C09103=1053.163,-16.101,428.307,170.734,30.867,155.806
C09104=1053.169,-15.852,428.293,170.735,30.869,155.806
C09105=1053.175,-15.602,428.279,170.737,30.871,155.806
C09106=1053.182,-15.353,428.265,170.739,30.873,155.807
C09107=1053.188,-15.103,428.251,170.741,30.875,155.807
C09108=1053.194,-14.853,428.238,170.742,30.877,155.807
C09109=1053.200,-14.604,428.223,170.744,30.878,155.807
C09110=1053.206,-14.354,428.209,170.746,30.880,155.808
C09111=1053.213,-14.104,428.195,170.747,30.882,155.808
C09112=1053.218,-13.855,428.181,170.749,30.884,155.808
C09113=1053.224,-13.606,428.167,170.751,30.886,155.808
C09114=1053.231,-13.356,428.153,170.753,30.888,155.809
C09115=1053.236,-13.107,428.139,170.755,30.890,155.809
C09116=1053.243,-12.857,428.124,170.756,30.892,155.809
C09117=1053.249,-12.608,428.110,170.758,30.894,155.809
C09118=1053.255,-12.358,428.095,170.759,30.896,155.810
C09119=1053.261,-12.109,428.082,170.761,30.898,155.810
C09120=1053.268,-11.859,428.067,170.763,30.900,155.810
C09121=1053.274,-11.610,428.053,170.765,30.902,155.810
C09122=1053.280,-11.360,428.038,170.767,30.903,155.810
C09123=1053.286,-11.111,428.025,170.768,30.905,155.811
C09124=1053.297,-10.694,428.001,170.771,30.909,155.811
C09125=1053.307,-10.278,427.977,170.774,30.912,155.812
C09126=1053.317,-9.862,427.954,170.777,30.915,155.812
C09127=1053.327,-9.446,427.930,170.780,30.918,155.812
C09128=1053.334,-9.196,427.915,170.781,30.920,155.813
C09129=1053.339,-8.946,427.901,170.782,30.922,155.813
C09130=1053.346,-8.697,427.887,170.784,30.925,155.813
C09131=1053.352,-8.447,427.873,170.786,30.926,155.813
C09132=1053.358,-8.198,427.858,170.788,30.928,155.814
C09133=1053.365,-7.949,427.844,170.790,30.930,155.814
C09134=1053.371,-7.699,427.830,170.792,30.932,155.814
C09135=1053.377,-7.449,427.815,170.793,30.934,155.814
C09136=1053.384,-7.201,427.801,170.794,30.936,155.815
C09137=1053.390,-6.950,427.786,170.796,30.938,155.815
C09138=1053.396,-6.701,427.772,170.798,30.940,155.815
C09139=1053.402,-6.452,427.757,170.800,30.942,155.816
C09140=1053.409,-6.202,427.743,170.802,30.944,155.816
C09141=1053.415,-5.953,427.729,170.804,30.946,155.816
C09142=1053.421,-5.703,427.714,170.804,30.947,155.816
C09143=1053.426,-5.453,427.700,170.806,30.950,155.817
C09144=1053.434,-5.204,427.686,170.808,30.952,155.817
C09145=1053.440,-4.954,427.671,170.810,30.954,155.817
C09146=1053.445,-4.705,427.657,170.812,30.955,155.817
C09147=1053.453,-4.456,427.642,170.814,30.957,155.818
C09148=1053.459,-4.206,427.627,170.815,30.960,155.818
C09149=1053.464,-3.956,427.614,170.816,30.962,155.818
C09150=1053.471,-3.707,427.599,170.818,30.963,155.818
C09151=1053.478,-3.457,427.584,170.820,30.965,155.819
C09152=1053.486,-3.092,427.563,170.823,30.968,155.819
C09153=1053.496,-2.727,427.541,170.825,30.971,155.819
C09154=1053.504,-2.362,427.520,170.827,30.974,155.820
C09155=1053.513,-1.997,427.498,170.830,30.977,155.820
C09156=1053.519,-1.747,427.484,170.831,30.979,155.821
C09157=1053.525,-1.497,427.469,170.833,30.981,155.821
C09158=1053.531,-1.248,427.454,170.835,30.983,155.821
C09159=1053.537,-0.998,427.439,170.837,30.986,155.821
C09160=1053.543,-0.749,427.425,170.838,30.988,155.822
C09161=1053.549,-0.500,427.410,170.840,30.990,155.822
C09162=1053.556,-0.250,427.395,170.841,30.992,155.822
C09163=1053.562,-0.001,427.380,170.843,30.994,155.823
C09164=1053.568,0.249,427.366,170.845,30.995,155.823
C09165=1053.574,0.499,427.351,170.847,30.998,155.823
C09166=1053.580,0.748,427.336,170.849,31.000,155.823
C09167=1053.586,0.998,427.321,170.849,31.002,155.824
C09168=1053.593,1.247,427.306,170.851,31.004,155.824
C09169=1053.598,1.496,427.292,170.853,31.006,155.824
C09170=1053.605,1.746,427.277,170.855,31.008,155.824
C09171=1053.611,1.996,427.262,170.857,31.010,155.825
C09172=1053.617,2.244,427.247,170.858,31.012,155.825
C09173=1053.623,2.494,427.232,170.859,31.014,155.825
C09174=1053.630,2.744,427.218,170.861,31.016,155.826
C09175=1053.636,2.993,427.203,170.863,31.018,155.826
C09176=1053.642,3.242,427.188,170.865,31.021,155.826
C09177=1053.648,3.492,427.173,170.866,31.023,155.826
C09178=1053.654,3.742,427.157,170.868,31.025,155.827
C09179=1053.660,3.991,427.143,170.870,31.026,155.827
C09180=1053.666,4.241,427.128,170.871,31.028,155.827
C09181=1053.672,4.490,427.113,170.873,31.030,155.827
C09182=1053.679,4.740,427.098,170.874,31.032,155.828
C09183=1053.685,4.989,427.083,170.876,31.035,155.828
C09184=1053.691,5.239,427.069,170.878,31.037,155.828
C09185=1053.697,5.488,427.054,170.880,31.039,155.829
C09186=1053.704,5.738,427.039,170.882,31.041,155.829
C09187=1053.709,5.987,427.024,170.882,31.043,155.829
C09188=1053.716,6.236,427.009,170.884,31.045,155.830
C09189=1053.722,6.486,426.994,170.886,31.047,155.830
C09190=1053.728,6.736,426.979,170.888,31.049,155.830
C09191=1053.734,6.986,426.964,170.890,31.051,155.830
C09192=1053.740,7.234,426.948,170.891,31.053,155.831
C09193=1053.747,7.484,426.933,170.893,31.055,155.831
C09194=1053.753,7.733,426.919,170.894,31.058,155.831
C09195=1053.759,7.983,426.904,170.896,31.060,155.832
C09196=1053.766,8.233,426.889,170.897,31.061,155.832
C09197=1053.772,8.482,426.874,170.899,31.063,155.832
C09198=1053.778,8.731,426.859,170.901,31.065,155.832
C09199=1053.784,8.981,426.843,170.903,31.067,155.833
C09200=1053.790,9.230,426.828,170.905,31.070,155.833
C09201=1053.797,9.480,426.813,170.905,31.072,155.833
C09202=1053.803,9.729,426.798,170.907,31.074,155.833
C09203=1053.809,9.979,426.783,170.909,31.076,155.834
C09204=1053.816,10.228,426.768,170.911,31.078,155.834
C09205=1053.822,10.477,426.753,170.913,31.080,155.834
C09206=1053.828,10.727,426.738,170.914,31.082,155.835
C09207=1053.834,10.977,426.722,170.916,31.084,155.835
C09208=1053.840,11.227,426.707,170.917,31.086,155.835
C09209=1053.846,11.475,426.692,170.919,31.088,155.835
C09210=1053.853,11.725,426.677,170.920,31.090,155.836
C09211=1053.859,11.974,426.662,170.922,31.092,155.836
C09212=1053.866,12.224,426.647,170.924,31.095,155.836
C09213=1053.872,12.473,426.632,170.926,31.097,155.837
C09214=1053.878,12.723,426.616,170.928,31.099,155.837
C09215=1053.884,12.973,426.601,170.928,31.100,155.837
C09216=1053.891,13.257,426.584,170.930,31.103,155.838
C09217=1053.899,13.541,426.566,170.932,31.105,155.838
C09218=1053.906,13.825,426.549,170.934,31.108,155.838
C09219=1053.913,14.110,426.532,170.936,31.110,155.838
C09220=1053.920,14.359,426.517,170.938,31.112,155.839
C09221=1053.925,14.609,426.501,170.939,31.114,155.839
C09222=1053.932,14.858,426.486,170.941,31.116,155.839
C09223=1053.939,15.107,426.470,170.943,31.118,155.840
C09224=1053.944,15.357,426.455,170.944,31.120,155.840
C09225=1053.950,15.606,426.440,170.946,31.122,155.840
C09226=1053.957,15.855,426.424,170.948,31.124,155.841
C09227=1053.962,16.105,426.409,170.950,31.127,155.841
C09228=1053.969,16.354,426.393,170.950,31.129,155.841
C09229=1053.975,16.604,426.377,170.952,31.131,155.842
C09230=1053.981,16.854,426.362,170.954,31.133,155.842
C09231=1053.988,17.103,426.347,170.956,31.135,155.842
C09232=1053.993,17.353,426.331,170.957,31.137,155.842
C09233=1054.000,17.602,426.316,170.959,31.140,155.843
C09234=1054.006,17.852,426.300,170.961,31.142,155.843
C09235=1054.012,18.100,426.285,170.962,31.144,155.843
C09236=1054.018,18.350,426.270,170.963,31.146,155.844
C09237=1054.024,18.599,426.254,170.965,31.148,155.844
C09238=1054.031,18.849,426.239,170.967,31.150,155.844
C09239=1054.036,19.098,426.222,170.969,31.153,155.845
C09240=1054.043,19.348,426.207,170.970,31.155,155.845
C09241=1054.050,19.597,426.192,170.972,31.157,155.845
C09242=1054.055,19.847,426.176,170.973,31.159,155.845
C09243=1054.062,20.096,426.161,170.975,31.161,155.846
C09244=1054.068,20.346,426.145,170.976,31.163,155.846
C09245=1054.074,20.595,426.129,170.978,31.165,155.846
C09246=1054.080,20.845,426.114,170.980,31.167,155.847
C09247=1054.087,21.094,426.098,170.982,31.169,155.847
C09248=1054.092,21.343,426.082,170.983,31.172,155.847
C09249=1054.099,21.593,426.067,170.984,31.174,155.848
C09250=1054.105,21.842,426.051,170.986,31.176,155.848
C09251=1054.110,22.092,426.035,170.988,31.178,155.848
C09252=1054.117,22.341,426.019,170.989,31.180,155.848
C09253=1054.123,22.591,426.003,170.991,31.182,155.849
C09254=1054.129,22.840,425.988,170.993,31.184,155.849
C09255=1054.135,23.090,425.972,170.995,31.187,155.849
C09256=1054.142,23.339,425.957,170.995,31.189,155.850
C09257=1054.148,23.589,425.941,170.997,31.191,155.850
C09258=1054.154,23.838,425.925,170.999,31.193,155.850
C09259=1054.160,24.088,425.910,171.000,31.195,155.851
C09260=1054.167,24.337,425.894,171.002,31.197,155.851
C09261=1054.173,24.586,425.878,171.004,31.199,155.851
C09262=1054.178,24.836,425.862,171.006,31.202,155.852
C09263=1054.185,25.085,425.846,171.007,31.204,155.852
C09264=1054.191,25.334,425.830,171.008,31.206,155.852
C09265=1054.198,25.584,425.815,171.010,31.208,155.852
C09266=1054.203,25.833,425.799,171.012,31.210,155.853
C09267=1054.210,26.083,425.783,171.013,31.212,155.853
C09268=1054.216,26.332,425.767,171.015,31.215,155.853
C09269=1054.222,26.581,425.751,171.017,31.217,155.854
C09270=1054.228,26.831,425.736,171.019,31.219,155.854
C09271=1054.234,27.080,425.720,171.019,31.221,155.854
C09272=1054.241,27.329,425.704,171.021,31.223,155.855
C09273=1054.247,27.579,425.688,171.023,31.226,155.855
C09274=1054.253,27.829,425.672,171.024,31.228,155.855
C09275=1054.260,28.078,425.656,171.026,31.230,155.856
C09276=1054.266,28.328,425.640,171.028,31.232,155.856
C09277=1054.272,28.577,425.624,171.030,31.234,155.856
C09278=1054.278,28.826,425.608,171.030,31.236,155.857
C09279=1054.284,29.076,425.592,171.032,31.238,155.857
C09280=1054.291,29.362,425.574,171.034,31.241,155.857
C09281=1054.298,29.646,425.555,171.036,31.244,155.858
C09282=1054.305,29.933,425.537,171.038,31.247,155.858
C09283=1054.312,30.218,425.518,171.040,31.249,155.858
C09284=1054.318,30.468,425.502,171.041,31.251,155.859
C09285=1054.324,30.717,425.486,171.042,31.253,155.859
C09286=1054.330,30.967,425.471,171.044,31.255,155.859
C09287=1054.336,31.216,425.455,171.046,31.258,155.860
C09288=1054.342,31.465,425.438,171.048,31.260,155.860
C09289=1054.348,31.715,425.422,171.049,31.262,155.860
C09290=1054.355,31.964,425.406,171.051,31.264,155.861
C09291=1054.362,32.214,425.390,171.053,31.266,155.861
C09292=1054.368,32.463,425.373,171.053,31.269,155.861
C09293=1054.373,32.712,425.357,171.055,31.271,155.862
C09294=1054.379,32.962,425.341,171.057,31.273,155.862
C09295=1054.386,33.211,425.325,171.059,31.275,155.862
C09296=1054.392,33.460,425.309,171.060,31.278,155.863
C09297=1054.398,33.709,425.293,171.062,31.280,155.863
C09298=1054.404,33.959,425.277,171.064,31.282,155.863
C09299=1054.411,34.209,425.260,171.064,31.284,155.864
C09300=1054.416,34.458,425.244,171.066,31.286,155.864
C09301=1054.423,34.707,425.228,171.068,31.289,155.864
C09302=1054.429,34.957,425.212,171.070,31.291,155.865
C09303=1054.435,35.206,425.195,171.071,31.293,155.865
C09304=1054.441,35.455,425.179,171.073,31.295,155.865
C09305=1054.448,35.705,425.163,171.075,31.298,155.866
C09306=1054.454,35.954,425.147,171.076,31.300,155.866
C09307=1054.460,36.204,425.131,171.077,31.302,155.866
C09308=1054.466,36.453,425.114,171.079,31.304,155.866
C09309=1054.472,36.702,425.098,171.081,31.307,155.867
C09310=1054.479,36.953,425.082,171.082,31.308,155.867
C09311=1054.485,37.202,425.065,171.084,31.311,155.867
C09312=1054.491,37.451,425.048,171.086,31.313,155.868
C09313=1054.498,37.700,425.033,171.087,31.315,155.868
C09314=1054.504,37.949,425.016,171.088,31.317,155.868
C09315=1054.510,38.199,425.000,171.090,31.319,155.869
C09316=1054.516,38.448,424.984,171.092,31.322,155.869
C09317=1054.522,38.698,424.967,171.093,31.324,155.869
C09318=1054.528,38.947,424.951,171.095,31.326,155.870
C09319=1054.533,39.196,424.933,171.097,31.329,155.870
C09320=1054.539,39.445,424.917,171.098,31.331,155.870
C09321=1054.546,39.696,424.901,171.099,31.333,155.871
C09322=1054.552,39.945,424.884,171.101,31.336,155.871
C09323=1054.558,40.194,424.868,171.102,31.338,155.871
C09324=1054.564,40.443,424.851,171.104,31.340,155.872
C09325=1054.571,40.693,424.834,171.106,31.342,155.872
C09326=1054.577,40.942,424.818,171.108,31.344,155.872
C09327=1054.583,41.192,424.802,171.109,31.346,155.873
C09328=1054.589,41.441,424.786,171.111,31.349,155.873
C09329=1054.595,41.690,424.769,171.112,31.351,155.873
C09330=1054.601,41.940,424.752,171.113,31.353,155.874
C09331=1054.607,42.189,424.736,171.115,31.355,155.874
C09332=1054.613,42.438,424.720,171.117,31.358,155.874
C09333=1054.619,42.687,424.703,171.118,31.360,155.875
C09334=1054.626,42.937,424.686,171.120,31.362,155.875
C09335=1054.632,43.187,424.670,171.122,31.365,155.875
C09336=1054.638,43.435,424.653,171.123,31.367,155.876
C09337=1054.644,43.685,424.637,171.124,31.369,155.876
C09338=1054.650,43.935,424.619,171.126,31.371,155.876
C09339=1054.656,44.184,424.602,171.128,31.374,155.877
C09340=1054.662,44.433,424.586,171.129,31.376,155.877
C09341=1054.667,44.683,424.569,171.131,31.378,155.877
C09342=1054.674,44.932,424.552,171.133,31.381,155.878
C09343=1054.680,45.182,424.536,171.134,31.383,155.878
C09344=1054.687,45.467,424.516,171.135,31.386,155.879
C09345=1054.694,45.753,424.497,171.137,31.388,155.879
C09346=1054.700,46.038,424.478,171.139,31.391,155.879
C09347=1054.708,46.324,424.458,171.141,31.394,155.880
C09348=1054.713,46.574,424.442,171.143,31.396,155.880
C09349=1054.720,46.822,424.425,171.144,31.398,155.881
C09350=1054.725,47.072,424.408,171.146,31.400,155.881
C09351=1054.732,47.321,424.390,171.147,31.403,155.881
C09352=1054.738,47.571,424.374,171.148,31.405,155.882
C09353=1054.744,47.819,424.357,171.150,31.408,155.882
C09354=1054.750,48.069,424.341,171.152,31.410,155.882
C09355=1054.756,48.319,424.324,171.153,31.412,155.883
C09356=1054.762,48.568,424.307,171.155,31.414,155.883
C09357=1054.768,48.817,424.290,171.157,31.417,155.883
C09358=1054.774,49.067,424.273,171.158,31.419,155.884
C09359=1054.780,49.316,424.256,171.159,31.421,155.884
C09360=1054.786,49.565,424.239,171.161,31.424,155.884
C09361=1054.792,49.815,424.221,171.163,31.426,155.885
C09362=1054.798,50.064,424.205,171.164,31.428,155.885
C09363=1054.804,50.313,424.188,171.166,31.431,155.885
C09364=1054.810,50.563,424.171,171.168,31.433,155.886
C09365=1054.817,50.812,424.154,171.169,31.435,155.886
C09366=1054.822,51.061,424.138,171.170,31.437,155.886
C09367=1054.829,51.311,424.120,171.172,31.440,155.887
C09368=1054.835,51.560,424.104,171.173,31.442,155.887
C09369=1054.841,51.809,424.087,171.175,31.444,155.887
C09370=1054.847,52.059,424.069,171.177,31.447,155.888
C09371=1054.853,52.308,424.052,171.178,31.449,155.888
C09372=1054.860,52.558,424.035,171.180,31.451,155.889
C09373=1054.865,52.807,424.018,171.182,31.453,155.889
C09374=1054.871,53.056,424.001,171.182,31.455,155.889
C09375=1054.878,53.305,423.984,171.184,31.458,155.890
C09376=1054.883,53.555,423.967,171.186,31.460,155.890
C09377=1054.890,53.805,423.950,171.187,31.463,155.890
C09378=1054.896,54.054,423.932,171.189,31.465,155.891
C09379=1054.902,54.303,423.916,171.191,31.467,155.891
C09380=1054.908,54.552,423.899,171.193,31.470,155.891
C09381=1054.914,54.801,423.881,171.194,31.471,155.892
C09382=1054.921,55.051,423.864,171.195,31.474,155.892
C09383=1054.927,55.300,423.847,171.197,31.476,155.892
C09384=1054.932,55.549,423.830,171.198,31.478,155.893
C09385=1054.939,55.799,423.813,171.200,31.481,155.893
C09386=1054.944,56.048,423.796,171.202,31.483,155.893
C09387=1054.951,56.298,423.778,171.203,31.486,155.894
C09388=1054.957,56.546,423.761,171.205,31.488,155.894
C09389=1054.963,56.797,423.744,171.207,31.490,155.894
C09390=1054.970,57.046,423.727,171.207,31.492,155.895
C09391=1054.976,57.295,423.710,171.209,31.494,155.895
C09392=1054.982,57.544,423.692,171.211,31.497,155.895
C09393=1054.988,57.794,423.676,171.212,31.499,155.896
C09394=1054.994,58.043,423.658,171.214,31.501,155.896
C09395=1055.001,58.293,423.641,171.216,31.504,155.896
C09396=1055.007,58.541,423.624,171.218,31.506,155.897
C09397=1055.013,58.792,423.606,171.219,31.508,155.897
C09398=1055.019,59.040,423.590,171.220,31.510,155.898
C09399=1055.025,59.290,423.572,171.222,31.513,155.898
C09400=1055.032,59.539,423.555,171.223,31.515,155.898
C09401=1055.038,59.788,423.537,171.225,31.517,155.899
C09402=1055.044,60.037,423.520,171.227,31.519,155.899
C09403=1055.050,60.287,423.503,171.228,31.522,155.899
C09404=1055.056,60.536,423.486,171.230,31.524,155.900
C09405=1055.063,60.786,423.468,171.232,31.526,155.900
C09406=1055.068,61.035,423.451,171.233,31.528,155.900
C09407=1055.075,61.284,423.433,171.234,31.531,155.901
C09408=1055.082,61.570,423.414,171.236,31.533,155.901
C09409=1055.090,61.855,423.394,171.238,31.536,155.901
C09410=1055.097,62.140,423.374,171.240,31.539,155.902
C09411=1055.104,62.425,423.355,171.242,31.541,155.902
C09412=1055.110,62.675,423.337,171.244,31.543,155.902
C09413=1055.116,62.924,423.320,171.245,31.545,155.903
C09414=1055.122,63.174,423.302,171.247,31.547,155.903
C09415=1055.129,63.423,423.284,171.248,31.550,155.904
C09416=1055.135,63.672,423.267,171.249,31.552,155.904
C09417=1055.141,63.921,423.250,171.251,31.555,155.904
C09418=1055.147,64.170,423.232,171.253,31.557,155.905
C09419=1055.154,64.420,423.215,171.254,31.559,155.905
C09420=1055.159,64.669,423.197,171.256,31.561,155.905
C09421=1055.165,64.919,423.179,171.258,31.563,155.906
C09422=1055.172,65.168,423.162,171.259,31.566,155.906
C09423=1055.178,65.417,423.144,171.260,31.568,155.906
C09424=1055.184,65.667,423.126,171.262,31.571,155.907
C09425=1055.190,65.916,423.109,171.263,31.573,155.907
C09426=1055.196,66.165,423.091,171.265,31.575,155.907
C09427=1055.202,66.414,423.074,171.267,31.577,155.908
C09428=1055.209,66.664,423.057,171.269,31.580,155.908
C09429=1055.214,66.913,423.039,171.270,31.582,155.908
C09430=1055.220,67.163,423.021,171.272,31.585,155.909
C09431=1055.227,67.411,423.003,171.273,31.587,155.909
C09432=1055.233,67.660,422.985,171.274,31.589,155.910
C09433=1055.239,67.910,422.967,171.276,31.591,155.910
C09434=1055.245,68.159,422.950,171.278,31.594,155.910
C09435=1055.252,68.409,422.933,171.279,31.596,155.911
C09436=1055.258,68.658,422.915,171.281,31.598,155.911
C09437=1055.263,68.907,422.897,171.283,31.601,155.911
C09438=1055.269,69.157,422.879,171.284,31.603,155.912
C09439=1055.276,69.405,422.861,171.286,31.605,155.912
C09440=1055.282,69.655,422.844,171.287,31.607,155.912
C09441=1055.288,69.905,422.826,171.288,31.610,155.913
C09442=1055.294,70.154,422.808,171.290,31.612,155.913
C09443=1055.300,70.404,422.790,171.292,31.615,155.913
C09444=1055.306,70.652,422.772,171.293,31.617,155.914
C09445=1055.312,70.901,422.754,171.295,31.619,155.914
C09446=1055.319,71.151,422.737,171.297,31.622,155.915
C09447=1055.324,71.400,422.719,171.298,31.624,155.915
C09448=1055.330,71.650,422.701,171.299,31.627,155.915
C09449=1055.336,71.898,422.683,171.301,31.629,155.916
C09450=1055.342,72.148,422.665,171.302,31.631,155.916
C09451=1055.348,72.398,422.647,171.304,31.633,155.916
C09452=1055.355,72.646,422.629,171.306,31.636,155.917
C09453=1055.361,72.896,422.611,171.307,31.638,155.917
C09454=1055.367,73.145,422.593,171.309,31.641,155.917
C09455=1055.373,73.395,422.576,171.311,31.643,155.918
C09456=1055.379,73.644,422.557,171.312,31.645,155.918
C09457=1055.385,73.893,422.539,171.313,31.647,155.919
C09458=1055.391,74.142,422.522,171.315,31.650,155.919
C09459=1055.397,74.392,422.503,171.317,31.652,155.919
C09460=1055.403,74.641,422.485,171.318,31.655,155.920
C09461=1055.409,74.890,422.467,171.320,31.657,155.920
C09462=1055.415,75.139,422.449,171.322,31.659,155.920
C09463=1055.421,75.389,422.431,171.323,31.661,155.921
C09464=1055.427,75.638,422.414,171.325,31.664,155.921
C09465=1055.434,75.887,422.395,171.327,31.666,155.921
C09466=1055.440,76.137,422.377,171.327,31.669,155.922
C09467=1055.446,76.385,422.359,171.329,31.671,155.922
C09468=1055.452,76.635,422.341,171.331,31.673,155.923
C09469=1055.458,76.885,422.323,171.332,31.676,155.923
C09470=1055.465,77.134,422.305,171.334,31.678,155.923
C09471=1055.470,77.383,422.287,171.336,31.681,155.924
C09472=1055.477,77.668,422.266,171.338,31.683,155.924
C09473=1055.484,77.954,422.245,171.340,31.686,155.924
C09474=1055.491,78.239,422.224,171.341,31.688,155.925
C09475=1055.498,78.524,422.204,171.342,31.691,155.925
C09476=1055.504,78.773,422.185,171.344,31.693,155.926
C09477=1055.510,79.023,422.167,171.346,31.696,155.926
C09478=1055.516,79.271,422.149,171.347,31.698,155.926
C09479=1055.522,79.521,422.131,171.349,31.700,155.927
C09480=1055.528,79.770,422.112,171.351,31.703,155.927
C09481=1055.534,80.019,422.093,171.352,31.705,155.928
C09482=1055.540,80.268,422.076,171.354,31.708,155.928
C09483=1055.546,80.517,422.057,171.355,31.710,155.928
C09484=1055.552,80.767,422.039,171.356,31.712,155.929
C09485=1055.558,81.016,422.020,171.358,31.715,155.929
C09486=1055.564,81.266,422.002,171.360,31.717,155.929
C09487=1055.570,81.515,421.984,171.362,31.720,155.930
C09488=1055.576,81.764,421.966,171.363,31.722,155.930
C09489=1055.582,82.013,421.948,171.365,31.724,155.931
C09490=1055.588,82.262,421.929,171.367,31.727,155.931
C09491=1055.594,82.512,421.910,171.368,31.729,155.931
C09492=1055.600,82.761,421.892,171.369,31.731,155.932
C09493=1055.606,83.010,421.874,171.371,31.734,155.932
C09494=1055.612,83.259,421.856,171.372,31.736,155.932
C09495=1055.619,83.508,421.837,171.374,31.739,155.933
C09496=1055.624,83.759,421.818,171.376,31.741,155.933
C09497=1055.630,84.008,421.800,171.377,31.743,155.934
C09498=1055.636,84.256,421.781,171.379,31.745,155.934
C09499=1055.642,84.506,421.763,171.381,31.748,155.934
C09500=1055.649,84.755,421.745,171.382,31.751,155.935
C09501=1055.654,85.004,421.726,171.384,31.753,155.935
C09502=1055.661,85.254,421.708,171.385,31.755,155.935
C09503=1055.666,85.503,421.689,171.386,31.757,155.936
C09504=1055.673,85.752,421.671,171.388,31.760,155.936
C09505=1055.679,86.001,421.652,171.390,31.762,155.936
C09506=1055.685,86.251,421.634,171.392,31.765,155.937
C09507=1055.691,86.500,421.615,171.393,31.767,155.937
C09508=1055.697,86.748,421.597,171.395,31.769,155.938
C09509=1055.703,86.997,421.578,171.397,31.772,155.938
C09510=1055.709,87.248,421.559,171.398,31.774,155.938
C09511=1055.715,87.497,421.541,171.399,31.776,155.939
C09512=1055.722,87.746,421.522,171.401,31.779,155.939
C09513=1055.728,87.995,421.504,171.402,31.781,155.939
C09514=1055.734,88.245,421.486,171.404,31.783,155.940
C09515=1055.739,88.493,421.467,171.406,31.786,155.940
C09516=1055.746,88.742,421.448,171.408,31.788,155.941
C09517=1055.752,88.992,421.429,171.409,31.790,155.941
C09518=1055.758,89.241,421.411,171.411,31.793,155.941
C09519=1055.764,89.491,421.392,171.413,31.795,155.942
C09520=1055.770,89.740,421.374,171.414,31.798,155.942
C09521=1055.777,89.989,421.355,171.415,31.800,155.942
C09522=1055.783,90.238,421.336,171.417,31.802,155.943
C09523=1055.789,90.488,421.317,171.418,31.804,155.943
C09524=1055.795,90.736,421.299,171.420,31.807,155.943
C09525=1055.800,90.985,421.280,171.422,31.810,155.944
C09526=1055.807,91.235,421.261,171.423,31.811,155.944
C09527=1055.812,91.485,421.242,171.425,31.814,155.945
C09528=1055.819,91.734,421.224,171.427,31.817,155.945
C09529=1055.825,91.983,421.205,171.429,31.819,155.945
C09530=1055.831,92.232,421.186,171.430,31.821,155.946
C09531=1055.837,92.481,421.167,171.431,31.824,155.946
C09532=1055.842,92.730,421.148,171.433,31.826,155.947
C09533=1055.849,92.979,421.130,171.434,31.829,155.947
C09534=1055.854,93.229,421.110,171.436,31.831,155.947
C09535=1055.861,93.478,421.092,171.438,31.833,155.948
C09536=1055.868,93.763,421.070,171.440,31.836,155.948
C09537=1055.874,94.048,421.048,171.442,31.839,155.949
C09538=1055.881,94.333,421.027,171.444,31.842,155.949
C09539=1055.888,94.618,421.005,171.445,31.844,155.949
C09540=1055.894,94.868,420.986,171.446,31.847,155.950
C09541=1055.900,95.117,420.967,171.448,31.849,155.950
C09542=1055.906,95.366,420.948,171.450,31.852,155.951
C09543=1055.912,95.616,420.929,171.451,31.854,155.951
C09544=1055.918,95.865,420.910,171.453,31.856,155.951
C09545=1055.924,96.114,420.891,171.455,31.859,155.952
C09546=1055.931,96.363,420.872,171.456,31.861,155.952
C09547=1055.936,96.613,420.853,171.458,31.864,155.952
C09548=1055.942,96.861,420.835,171.460,31.866,155.953
C09549=1055.948,97.110,420.815,171.462,31.868,155.953
C09550=1055.955,97.359,420.796,171.462,31.871,155.954
C09551=1055.960,97.608,420.777,171.464,31.873,155.954
C09552=1055.967,97.858,420.758,171.466,31.875,155.954
C09553=1055.972,98.107,420.739,171.467,31.878,155.955
C09554=1055.978,98.356,420.720,171.469,31.880,155.955
C09555=1055.984,98.606,420.701,171.471,31.883,155.956
C09556=1055.990,98.855,420.682,171.473,31.885,155.956
C09557=1055.997,99.103,420.662,171.474,31.887,155.956
C09558=1056.003,99.353,420.643,171.476,31.890,155.957
C09559=1056.009,99.602,420.625,171.478,31.892,155.957
C09560=1056.015,99.851,420.605,171.478,31.894,155.957
C09561=1056.021,100.101,420.587,171.480,31.897,155.958
C09562=1056.027,100.350,420.567,171.482,31.899,155.958
C09563=1056.033,100.600,420.547,171.484,31.902,155.959
C09564=1056.040,100.849,420.528,171.485,31.904,155.959
C09565=1056.045,101.098,420.509,171.487,31.906,155.959
C09566=1056.051,101.348,420.490,171.489,31.909,155.960
C09567=1056.058,101.596,420.471,171.490,31.911,155.960
C09568=1056.064,101.845,420.451,171.492,31.914,155.960
C09569=1056.069,102.095,420.432,171.494,31.916,155.961
C09570=1056.075,102.344,420.412,171.495,31.919,155.961
C09571=1056.081,102.593,420.393,171.496,31.921,155.962
C09572=1056.087,102.842,420.374,171.498,31.923,155.962
C09573=1056.093,103.092,420.355,171.500,31.926,155.962
C09574=1056.099,103.340,420.335,171.501,31.928,155.963
C09575=1056.105,103.590,420.316,171.503,31.931,155.963
C09576=1056.111,103.839,420.297,171.505,31.933,155.964
C09577=1056.117,104.088,420.277,171.507,31.935,155.964
C09578=1056.123,104.337,420.258,171.508,31.938,155.964
C09579=1056.129,104.586,420.238,171.510,31.941,155.965
C09580=1056.135,104.836,420.219,171.512,31.943,155.965
C09581=1056.141,105.085,420.200,171.512,31.945,155.965
C09582=1056.147,105.333,420.180,171.514,31.948,155.966
C09583=1056.153,105.583,420.161,171.516,31.950,155.966
C09584=1056.158,105.832,420.142,171.518,31.952,155.967
C09585=1056.164,106.081,420.122,171.519,31.955,155.967
C09586=1056.171,106.330,420.103,171.521,31.958,155.967
C09587=1056.177,106.579,420.083,171.523,31.960,155.968
C09588=1056.182,106.829,420.064,171.525,31.962,155.968
C09589=1056.188,107.077,420.044,171.526,31.965,155.969
C09590=1056.195,107.327,420.024,171.528,31.967,155.969
C09591=1056.201,107.576,420.004,171.530,31.969,155.969
C09592=1056.207,107.825,419.986,171.530,31.972,155.970
C09593=1056.213,108.075,419.966,171.532,31.974,155.970
C09594=1056.219,108.324,419.946,171.534,31.977,155.970
C09595=1056.224,108.573,419.927,171.536,31.979,155.971
C09596=1056.230,108.822,419.907,171.537,31.981,155.971
C09597=1056.236,109.071,419.888,171.539,31.984,155.972
C09598=1056.244,109.321,419.868,171.541,31.986,155.972
C09599=1056.250,109.569,419.848,171.543,31.989,155.972
C09600=1056.256,109.854,419.826,171.545,31.991,155.973
C09601=1056.262,110.140,419.804,171.547,31.994,155.973
C09602=1056.270,110.425,419.781,171.548,31.997,155.974
C09603=1056.277,110.710,419.759,171.550,32.000,155.974
C09604=1056.283,110.959,419.739,171.551,32.002,155.975
C09605=1056.289,111.208,419.720,171.553,32.004,155.975
C09606=1056.294,111.457,419.700,171.555,32.007,155.975
C09607=1056.301,111.707,419.680,171.557,32.010,155.976
C09608=1056.307,111.956,419.660,171.558,32.011,155.976
C09609=1056.313,112.205,419.641,171.560,32.014,155.976
C09610=1056.319,112.454,419.621,171.562,32.017,155.977
C09611=1056.325,112.703,419.601,171.564,32.019,155.977
C09612=1056.330,112.952,419.582,171.565,32.021,155.978
C09613=1056.337,113.202,419.561,171.567,32.024,155.978
C09614=1056.343,113.451,419.541,171.568,32.027,155.978
C09615=1056.349,113.700,419.522,171.570,32.029,155.979
C09616=1056.355,113.949,419.502,171.571,32.031,155.979
C09617=1056.361,114.198,419.482,171.573,32.034,155.980
C09618=1056.366,114.447,419.463,171.575,32.036,155.980
C09619=1056.372,114.697,419.442,171.577,32.039,155.980
C09620=1056.378,114.946,419.422,171.578,32.041,155.981
C09621=1056.384,115.194,419.402,171.580,32.044,155.981
C09622=1056.390,115.444,419.383,171.582,32.046,155.982
C09623=1056.396,115.693,419.363,171.584,32.049,155.982
C09624=1056.401,115.942,419.342,171.585,32.051,155.983
C09625=1056.407,116.191,419.322,171.586,32.054,155.983
C09626=1056.413,116.441,419.303,171.588,32.056,155.983
C09627=1056.419,116.690,419.283,171.590,32.059,155.984
C09628=1056.425,116.939,419.262,171.591,32.061,155.984
C09629=1056.431,117.188,419.242,171.593,32.064,155.985
C09630=1056.437,117.436,419.222,171.595,32.066,155.985
C09631=1056.443,117.686,419.202,171.597,32.068,155.985
C09632=1056.448,117.936,419.182,171.598,32.071,155.986
C09633=1056.454,118.184,419.162,171.600,32.074,155.986
C09634=1056.460,118.433,419.142,171.602,32.076,155.987
C09635=1056.466,118.682,419.122,171.604,32.079,155.987
C09636=1056.472,118.932,419.101,171.605,32.081,155.987
C09637=1056.478,119.181,419.081,171.606,32.083,155.988
C09638=1056.484,119.429,419.061,171.608,32.086,155.988
C09639=1056.490,119.678,419.041,171.610,32.089,155.989
C09640=1056.496,119.928,419.021,171.611,32.091,155.989
C09641=1056.502,120.178,419.001,171.613,32.093,155.989
C09642=1056.508,120.426,418.981,171.615,32.096,155.990
C09643=1056.514,120.675,418.961,171.617,32.098,155.990
C09644=1056.519,120.925,418.940,171.618,32.101,155.991
C09645=1056.525,121.174,418.921,171.620,32.104,155.991
C09646=1056.531,121.423,418.901,171.622,32.106,155.991
C09647=1056.537,121.672,418.880,171.624,32.108,155.992
C09648=1056.543,121.921,418.860,171.626,32.111,155.992
C09649=1056.549,122.170,418.840,171.626,32.113,155.993
C09650=1056.555,122.419,418.820,171.628,32.115,155.993
C09651=1056.561,122.669,418.799,171.630,32.118,155.993
C09652=1056.567,122.918,418.779,171.632,32.121,155.994
C09653=1056.573,123.166,418.759,171.633,32.123,155.994
C09654=1056.578,123.415,418.738,171.635,32.125,155.994
C09655=1056.585,123.665,418.718,171.637,32.128,155.995
C09656=1056.591,123.914,418.698,171.639,32.130,155.995
C09657=1056.596,124.163,418.678,171.641,32.133,155.996
C09658=1056.603,124.412,418.657,171.642,32.136,155.996
C09659=1056.609,124.661,418.637,171.644,32.138,155.996
C09660=1056.615,124.909,418.617,171.646,32.140,155.997
C09661=1056.621,125.159,418.596,171.647,32.143,155.997
C09662=1056.627,125.408,418.576,171.649,32.145,155.998
C09663=1056.633,125.657,418.556,171.650,32.147,155.998
C09664=1056.640,125.942,418.532,171.652,32.151,155.999
C09665=1056.647,126.228,418.508,171.654,32.153,155.999
C09666=1056.653,126.512,418.485,171.657,32.156,155.999
C09667=1056.660,126.798,418.461,171.659,32.159,156.000
C09668=1056.666,127.047,418.442,171.660,32.161,156.000
C09669=1056.672,127.295,418.422,171.662,32.164,156.001
C09670=1056.678,127.545,418.401,171.664,32.166,156.001
C09671=1056.684,127.794,418.381,171.666,32.168,156.001
C09672=1056.691,128.043,418.360,171.668,32.171,156.002
C09673=1056.696,128.292,418.339,171.668,32.173,156.002
C09674=1056.702,128.541,418.319,171.670,32.176,156.003
C09675=1056.709,128.790,418.299,171.672,32.178,156.003
C09676=1056.714,129.039,418.278,171.674,32.181,156.003
C09677=1056.721,129.288,418.257,171.676,32.183,156.004
C09678=1056.727,129.537,418.237,171.678,32.185,156.004
C09679=1056.733,129.787,418.216,171.679,32.188,156.005
C09680=1056.739,130.036,418.196,171.681,32.191,156.005
C09681=1056.745,130.284,418.176,171.683,32.193,156.005
C09682=1056.751,130.534,418.155,171.685,32.195,156.006
C09683=1056.757,130.783,418.135,171.687,32.198,156.006
C09684=1056.764,131.032,418.115,171.689,32.200,156.007
C09685=1056.769,131.281,418.093,171.690,32.202,156.007
C09686=1056.776,131.530,418.073,171.692,32.205,156.007
C09687=1056.781,131.779,418.052,171.693,32.208,156.008
C09688=1056.788,132.028,418.031,171.695,32.210,156.008
C09689=1056.793,132.277,418.011,171.697,32.213,156.009
C09690=1056.799,132.527,417.989,171.699,32.215,156.009
C09691=1056.805,132.775,417.969,171.700,32.217,156.009
C09692=1056.811,133.024,417.949,171.702,32.220,156.010
C09693=1056.818,133.273,417.928,171.704,32.223,156.010
C09694=1056.823,133.522,417.907,171.706,32.225,156.011
C09695=1056.829,133.772,417.885,171.708,32.228,156.011
C09696=1056.835,134.021,417.865,171.709,32.230,156.012
C09697=1056.841,134.270,417.845,171.711,32.233,156.012
C09698=1056.846,134.519,417.823,171.713,32.235,156.012
C09699=1056.853,134.768,417.803,171.715,32.238,156.013
C09700=1056.859,135.017,417.782,171.716,32.240,156.013
C09701=1056.864,135.266,417.761,171.718,32.243,156.014
C09702=1056.871,135.515,417.740,171.719,32.245,156.014
C09703=1056.876,135.764,417.719,171.721,32.248,156.014
C09704=1056.882,136.013,417.698,171.723,32.250,156.015
C09705=1056.888,136.262,417.678,171.725,32.252,156.015
C09706=1056.894,136.511,417.656,171.727,32.255,156.016
C09707=1056.899,136.760,417.636,171.729,32.258,156.016
C09708=1056.906,137.009,417.615,171.731,32.260,156.016
C09709=1056.912,137.258,417.594,171.732,32.263,156.017
C09710=1056.918,137.508,417.572,171.734,32.265,156.017
C09711=1056.924,137.756,417.553,171.736,32.267,156.018
C09712=1056.930,138.006,417.531,171.738,32.270,156.018
C09713=1056.936,138.255,417.509,171.740,32.273,156.018
C09714=1056.942,138.504,417.489,171.741,32.275,156.019
C09715=1056.948,138.753,417.468,171.743,32.278,156.019
C09716=1056.954,139.002,417.447,171.744,32.280,156.020
C09717=1056.960,139.251,417.425,171.746,32.282,156.020
C09718=1056.966,139.499,417.405,171.748,32.285,156.020
C09719=1056.972,139.749,417.384,171.750,32.288,156.021
C09720=1056.977,139.998,417.363,171.752,32.290,156.021
C09721=1056.984,140.247,417.341,171.754,32.293,156.022
C09722=1056.989,140.496,417.320,171.756,32.295,156.022
C09723=1056.995,140.745,417.299,171.757,32.298,156.023
C09724=1057.001,140.993,417.278,171.759,32.301,156.023
C09725=1057.007,141.243,417.257,171.761,32.303,156.023
C09726=1057.013,141.492,417.236,171.763,32.306,156.024
C09727=1057.019,141.741,417.214,171.765,32.308,156.024
C09728=1057.025,142.027,417.190,171.766,32.311,156.025
C09729=1057.032,142.311,417.166,171.768,32.314,156.025
C09730=1057.039,142.595,417.142,171.770,32.317,156.026
C09731=1057.046,142.881,417.117,171.772,32.319,156.026
C09732=1057.051,143.130,417.096,171.774,32.322,156.027
C09733=1057.057,143.379,417.075,171.776,32.325,156.027
C09734=1057.064,143.628,417.053,171.778,32.327,156.027
C09735=1057.070,143.876,417.032,171.780,32.330,156.028
C09736=1057.076,144.126,417.011,171.782,32.332,156.028
C09737=1057.081,144.375,416.990,171.784,32.335,156.029
C09738=1057.087,144.624,416.968,171.786,32.338,156.029
C09739=1057.093,144.873,416.947,171.787,32.340,156.030
C09740=1057.099,145.122,416.925,171.789,32.343,156.030
C09741=1057.105,145.371,416.904,171.791,32.345,156.030
C09742=1057.111,145.621,416.883,171.793,32.347,156.031
C09743=1057.117,145.869,416.862,171.794,32.350,156.031
C09744=1057.123,146.118,416.840,171.796,32.353,156.032
C09745=1057.129,146.367,416.818,171.798,32.355,156.032
C09746=1057.134,146.616,416.797,171.800,32.358,156.032
C09747=1057.141,146.865,416.775,171.802,32.360,156.033
C09748=1057.147,147.113,416.755,171.804,32.363,156.033
C09749=1057.153,147.363,416.733,171.805,32.366,156.034
C09750=1057.159,147.612,416.712,171.807,32.368,156.034
C09751=1057.165,147.860,416.690,171.809,32.371,156.035
C09752=1057.171,148.109,416.669,171.811,32.373,156.035
C09753=1057.176,148.359,416.646,171.813,32.376,156.035
C09754=1057.182,148.607,416.625,171.815,32.379,156.036
C09755=1057.188,148.857,416.603,171.817,32.381,156.036
C09756=1057.194,149.106,416.582,171.819,32.383,156.037
C09757=1057.200,149.354,416.561,171.821,32.386,156.037
C09758=1057.206,149.604,416.539,171.823,32.388,156.037
C09759=1057.212,149.853,416.517,171.824,32.391,156.038
C09760=1057.218,150.101,416.496,171.825,32.393,156.038
C09761=1057.224,150.351,416.474,171.827,32.396,156.039
C09762=1057.229,150.600,416.452,171.829,32.399,156.039
C09763=1057.235,150.849,416.431,171.831,32.401,156.040
C09764=1057.241,151.098,416.409,171.833,32.404,156.040
C09765=1057.247,151.347,416.388,171.835,32.406,156.040
C09766=1057.253,151.596,416.366,171.837,32.409,156.041
C09767=1057.259,151.845,416.345,171.839,32.412,156.041
C09768=1057.264,152.094,416.322,171.841,32.414,156.042
C09769=1057.270,152.343,416.301,171.843,32.417,156.042
C09770=1057.276,152.591,416.279,171.845,32.419,156.043
C09771=1057.283,152.840,416.257,171.847,32.422,156.043
C09772=1057.289,153.090,416.236,171.849,32.425,156.043
C09773=1057.295,153.339,416.214,171.851,32.427,156.044
C09774=1057.300,153.588,416.192,171.852,32.430,156.044
C09775=1057.306,153.837,416.170,171.854,32.432,156.045
C09776=1057.312,154.086,416.148,171.855,32.435,156.045
C09777=1057.318,154.335,416.126,171.857,32.438,156.046
C09778=1057.324,154.583,416.105,171.859,32.440,156.046
C09779=1057.329,154.833,416.083,171.861,32.443,156.046
C09780=1057.336,155.081,416.061,171.863,32.445,156.047
C09781=1057.342,155.331,416.039,171.865,32.448,156.047
C09782=1057.348,155.580,416.017,171.867,32.450,156.048
C09783=1057.353,155.829,415.996,171.869,32.453,156.048
C09784=1057.360,156.077,415.973,171.871,32.456,156.049
C09785=1057.366,156.326,415.952,171.873,32.458,156.049
C09786=1057.371,156.576,415.929,171.875,32.461,156.050
C09787=1057.377,156.824,415.908,171.877,32.464,156.050
C09788=1057.383,157.073,415.886,171.879,32.467,156.050
C09789=1057.389,157.322,415.863,171.881,32.469,156.051
C09790=1057.395,157.572,415.842,171.883,32.472,156.051
C09791=1057.401,157.820,415.819,171.885,32.474,156.052
C09792=1057.407,158.105,415.795,171.887,32.477,156.052
C09793=1057.414,158.389,415.769,171.888,32.480,156.053
C09794=1057.421,158.674,415.744,171.890,32.483,156.053
C09795=1057.428,158.959,415.719,171.893,32.486,156.054
C09796=1057.434,159.208,415.697,171.895,32.489,156.054
C09797=1057.439,159.457,415.674,171.897,32.491,156.054
C09798=1057.445,159.705,415.653,171.899,32.494,156.055
C09799=1057.451,159.954,415.630,171.901,32.496,156.055
C09800=1057.457,160.203,415.608,171.903,32.499,156.056
C09801=1057.463,160.453,415.586,171.905,32.502,156.056
C09802=1057.470,160.701,415.564,171.907,32.505,156.057
C09803=1057.475,160.951,415.542,171.909,32.507,156.057
C09804=1057.481,161.198,415.520,171.910,32.510,156.058
C09805=1057.486,161.448,415.498,171.912,32.512,156.058
C09806=1057.492,161.697,415.475,171.914,32.515,156.058
C09807=1057.498,161.946,415.452,171.916,32.518,156.059
C09808=1057.504,162.195,415.430,171.918,32.521,156.059
C09809=1057.509,162.443,415.408,171.920,32.523,156.060
C09810=1057.514,162.693,415.385,171.922,32.526,156.060
C09811=1057.521,162.941,415.363,171.923,32.529,156.061
C09812=1057.526,163.191,415.341,171.925,32.532,156.061
C09813=1057.532,163.440,415.318,171.927,32.534,156.062
C09814=1057.537,163.688,415.295,171.929,32.537,156.062
C09815=1057.543,163.937,415.274,171.931,32.540,156.063
C09816=1057.549,164.186,415.251,171.933,32.543,156.063
C09817=1057.555,164.435,415.228,171.935,32.545,156.064
C09818=1057.561,164.684,415.206,171.937,32.548,156.064
C09819=1057.567,164.933,415.183,171.939,32.550,156.064
C09820=1057.572,165.182,415.160,171.941,32.554,156.065
C09821=1057.577,165.431,415.138,171.943,32.556,156.065
C09822=1057.584,165.679,415.116,171.945,32.559,156.066
C09823=1057.589,165.928,415.093,171.947,32.561,156.066
C09824=1057.595,166.178,415.071,171.949,32.565,156.067
C09825=1057.601,166.427,415.048,171.951,32.567,156.067
C09826=1057.607,166.675,415.025,171.953,32.570,156.068
C09827=1057.613,166.924,415.003,171.955,32.572,156.068
C09828=1057.618,167.174,414.980,171.957,32.576,156.069
C09829=1057.624,167.423,414.957,171.959,32.578,156.069
C09830=1057.630,167.670,414.935,171.961,32.581,156.070
C09831=1057.636,167.919,414.912,171.963,32.583,156.070
C09832=1057.641,168.169,414.890,171.964,32.586,156.071
C09833=1057.647,168.418,414.867,171.966,32.589,156.071
C09834=1057.652,168.667,414.844,171.968,32.592,156.071
C09835=1057.659,168.915,414.822,171.970,32.594,156.072
C09836=1057.665,169.164,414.799,171.973,32.597,156.072
C09837=1057.670,169.414,414.777,171.975,32.600,156.073
C09838=1057.676,169.663,414.754,171.977,32.603,156.073
C09839=1057.682,169.911,414.731,171.979,32.605,156.074
C09840=1057.688,170.160,414.709,171.981,32.608,156.074
C09841=1057.694,170.409,414.686,171.983,32.611,156.075
C09842=1057.699,170.658,414.663,171.985,32.614,156.075
C09843=1057.705,170.907,414.640,171.987,32.616,156.075
C09844=1057.712,171.155,414.617,171.989,32.619,156.076
C09845=1057.717,171.404,414.594,171.991,32.622,156.076
C09846=1057.723,171.654,414.572,171.993,32.624,156.077
C09847=1057.729,171.903,414.549,171.995,32.627,156.077
C09848=1057.734,172.151,414.526,171.997,32.630,156.078
C09849=1057.741,172.400,414.504,171.999,32.633,156.078
C09850=1057.746,172.649,414.481,172.001,32.635,156.079
C09851=1057.752,172.898,414.458,172.003,32.638,156.079
C09852=1057.758,173.147,414.435,172.005,32.641,156.080
C09853=1057.764,173.396,414.412,172.007,32.644,156.080
C09854=1057.769,173.645,414.389,172.009,32.646,156.081
C09855=1057.776,173.893,414.367,172.011,32.649,156.081
C09856=1057.782,174.177,414.340,172.013,32.652,156.082
C09857=1057.789,174.462,414.314,172.015,32.655,156.082
C09858=1057.796,174.746,414.288,172.018,32.659,156.083
C09859=1057.803,175.030,414.262,172.020,32.661,156.083
C09860=1057.809,175.279,414.239,172.022,32.664,156.084
C09861=1057.815,175.528,414.216,172.024,32.667,156.084
C09862=1057.820,175.777,414.193,172.026,32.669,156.084
C09863=1057.826,176.026,414.170,172.029,32.672,156.085
C09864=1057.832,176.274,414.147,172.031,32.675,156.085
C09865=1057.838,176.523,414.124,172.033,32.678,156.086
C09866=1057.845,176.772,414.101,172.035,32.680,156.086
C09867=1057.851,177.021,414.078,172.037,32.683,156.087
C09868=1057.856,177.270,414.055,172.039,32.686,156.087
C09869=1057.862,177.519,414.032,172.041,32.689,156.088
C09870=1057.868,177.768,414.009,172.043,32.691,156.088
C09871=1057.874,178.017,413.986,172.045,32.694,156.089
C09872=1057.880,178.266,413.962,172.048,32.697,156.089
C09873=1057.887,178.514,413.940,172.050,32.700,156.090
C09874=1057.893,178.763,413.917,172.052,32.702,156.090
C09875=1057.898,179.012,413.894,172.054,32.705,156.090
C09876=1057.904,179.261,413.871,172.056,32.708,156.091
C09877=1057.910,179.509,413.847,172.058,32.711,156.091
C09878=1057.916,179.759,413.824,172.060,32.713,156.092
C09879=1057.922,180.008,413.801,172.061,32.716,156.092
C09880=1057.928,180.256,413.778,172.064,32.719,156.093
C09881=1057.934,180.505,413.755,172.066,32.722,156.093
C09882=1057.941,180.754,413.732,172.068,32.724,156.094
C09883=1057.947,181.003,413.709,172.070,32.727,156.094
C09884=1057.953,181.251,413.685,172.072,32.730,156.095
C09885=1057.958,181.500,413.662,172.074,32.732,156.095
C09886=1057.964,181.749,413.639,172.076,32.735,156.096
C09887=1057.971,181.998,413.615,172.079,32.738,156.096
C09888=1057.977,182.247,413.592,172.081,32.741,156.097
C09889=1057.982,182.496,413.569,172.083,32.743,156.097
C09890=1057.989,182.745,413.545,172.085,32.746,156.097
C09891=1057.995,182.994,413.522,172.087,32.749,156.098
C09892=1058.000,183.243,413.499,172.089,32.752,156.098
C09893=1058.006,183.491,413.476,172.092,32.754,156.099
C09894=1058.013,183.740,413.453,172.094,32.757,156.099
C09895=1058.020,183.988,413.429,172.096,32.760,156.100
C09896=1058.025,184.237,413.406,172.098,32.763,156.100
C09897=1058.032,184.487,413.383,172.100,32.765,156.101
C09898=1058.037,184.735,413.359,172.102,32.768,156.101
C09899=1058.043,184.984,413.336,172.105,32.771,156.102
C09900=1058.048,185.233,413.312,172.107,32.774,156.102
C09901=1058.054,185.481,413.288,172.109,32.777,156.103
C09902=1058.060,185.731,413.264,172.111,32.780,156.103
C09903=1058.066,185.979,413.240,172.113,32.782,156.104
C09904=1058.071,186.228,413.218,172.115,32.786,156.104
C09905=1058.077,186.477,413.193,172.118,32.789,156.105
C09906=1058.082,186.726,413.170,172.120,32.791,156.105
C09907=1058.088,186.975,413.146,172.122,32.795,156.106
C09908=1058.094,187.223,413.122,172.124,32.797,156.106
C09909=1058.100,187.472,413.099,172.126,32.800,156.107
C09910=1058.105,187.721,413.075,172.128,32.803,156.107
C09911=1058.112,187.970,413.051,172.130,32.806,156.108
C09912=1058.117,188.219,413.027,172.132,32.809,156.108
C09913=1058.123,188.467,413.004,172.134,32.812,156.109
C09914=1058.128,188.716,412.979,172.136,32.815,156.109
C09915=1058.135,188.965,412.956,172.138,32.818,156.110
C09916=1058.141,189.214,412.932,172.141,32.821,156.110
C09917=1058.146,189.462,412.908,172.143,32.823,156.111
C09918=1058.152,189.712,412.885,172.145,32.827,156.111
C09919=1058.158,189.961,412.861,172.147,32.829,156.112
C09920=1058.164,190.244,412.833,172.150,32.833,156.112
C09921=1058.172,190.528,412.806,172.152,32.836,156.113
C09922=1058.178,190.811,412.779,172.155,32.839,156.113
C09923=1058.185,191.096,412.752,172.157,32.842,156.114
C09924=1058.190,191.344,412.728,172.159,32.846,156.114
C09925=1058.196,191.592,412.704,172.162,32.849,156.115
C09926=1058.202,191.842,412.680,172.164,32.851,156.115
C09927=1058.208,192.091,412.656,172.166,32.855,156.116
C09928=1058.213,192.339,412.632,172.168,32.857,156.116
C09929=1058.220,192.588,412.608,172.171,32.860,156.117
C09930=1058.225,192.837,412.584,172.173,32.863,156.118
C09931=1058.231,193.085,412.560,172.175,32.866,156.118
C09932=1058.237,193.334,412.535,172.177,32.869,156.119
C09933=1058.243,193.583,412.513,172.179,32.872,156.119
C09934=1058.248,193.832,412.488,172.182,32.875,156.120
C09935=1058.255,194.081,412.464,172.184,32.878,156.120
C09936=1058.261,194.329,412.441,172.186,32.881,156.121
C09937=1058.266,194.578,412.416,172.188,32.884,156.121
C09938=1058.272,194.827,412.392,172.191,32.886,156.121
C09939=1058.278,195.076,412.368,172.193,32.890,156.122
C09940=1058.284,195.324,412.343,172.195,32.893,156.123
C09941=1058.290,195.573,412.319,172.197,32.895,156.123
C09942=1058.296,195.822,412.295,172.200,32.899,156.124
C09943=1058.302,196.070,412.271,172.202,32.901,156.124
C09944=1058.308,196.320,412.247,172.204,32.904,156.125
C09945=1058.314,196.568,412.223,172.207,32.907,156.125
C09946=1058.320,196.817,412.199,172.209,32.910,156.126
C09947=1058.326,197.065,412.175,172.211,32.913,156.126
C09948=1058.331,197.315,412.150,172.213,32.916,156.127
C09949=1058.337,197.563,412.127,172.216,32.919,156.127
C09950=1058.343,197.812,412.102,172.218,32.922,156.128
C09951=1058.349,198.061,412.078,172.220,32.925,156.128
C09952=1058.355,198.310,412.054,172.222,32.928,156.129
C09953=1058.361,198.558,412.030,172.225,32.931,156.129
C09954=1058.368,198.807,412.005,172.227,32.934,156.130
C09955=1058.374,199.055,411.981,172.229,32.937,156.130
C09956=1058.379,199.304,411.956,172.232,32.940,156.131
C09957=1058.385,199.554,411.932,172.234,32.942,156.131
C09958=1058.391,199.802,411.908,172.235,32.946,156.132
C09959=1058.397,200.051,411.884,172.238,32.949,156.132
C09960=1058.403,200.300,411.860,172.240,32.951,156.133
C09961=1058.410,200.548,411.835,172.242,32.955,156.133
C09962=1058.416,200.796,411.811,172.245,32.958,156.134
C09963=1058.422,201.046,411.786,172.247,32.960,156.134
C09964=1058.427,201.295,411.762,172.249,32.963,156.135
C09965=1058.434,201.543,411.737,172.251,32.967,156.135
C09966=1058.440,201.792,411.713,172.254,32.969,156.136
C09967=1058.446,202.040,411.689,172.256,32.972,156.136
C09968=1058.452,202.290,411.664,172.258,32.975,156.137
C09969=1058.457,202.537,411.639,172.261,32.979,156.137
C09970=1058.463,202.787,411.615,172.263,32.982,156.138
C09971=1058.468,203.035,411.590,172.265,32.984,156.138
C09972=1058.475,203.284,411.565,172.268,32.988,156.139
C09973=1058.481,203.533,411.541,172.270,32.991,156.140
C09974=1058.487,203.782,411.517,172.272,32.994,156.140
C09975=1058.493,204.030,411.492,172.275,32.997,156.141
C09976=1058.498,204.279,411.467,172.277,33.000,156.141
C09977=1058.504,204.528,411.442,172.279,33.003,156.142
C09978=1058.510,204.777,411.417,172.282,33.006,156.142
C09979=1058.515,205.025,411.393,172.284,33.009,156.143
C09980=1058.522,205.274,411.368,172.286,33.012,156.143
C09981=1058.528,205.522,411.344,172.289,33.015,156.144
C09982=1058.534,205.771,411.319,172.291,33.019,156.144
C09983=1058.540,206.020,411.294,172.293,33.022,156.145
C09984=1058.565,207.070,411.190,172.482,33.109,156.156
C09985=1058.574,207.456,411.150,172.485,33.115,156.157
C09986=1058.584,207.841,411.110,172.488,33.121,156.158
C09987=1058.594,208.228,411.069,172.491,33.127,156.159
C09988=1058.603,208.614,411.030,172.494,33.133,156.160
C09989=1058.610,208.863,411.005,172.497,33.137,156.161
C09990=1058.615,209.111,410.978,172.499,33.141,156.162
C09991=1058.622,209.360,410.953,172.500,33.145,156.163
C09992=1058.628,209.608,410.927,172.502,33.149,156.163
C09993=1058.634,209.856,410.901,172.504,33.153,156.164
C09994=1058.640,210.105,410.875,172.506,33.157,156.165
C09995=1058.646,210.353,410.849,172.508,33.161,156.166
C09996=1058.652,210.602,410.824,172.510,33.165,156.166
//INST
///DATE 2021/06/25 14:46
///ATTR SC,RW,RJ
////FRAME ROBOT
///GROUP1 RB1
NOP
MOVL C00000 V=800.0 PL=0
MOVL C00001 V=800.0 PL=0
MOVL C00002 V=800.0 PL=0
MOVL C00003 V=800.0 PL=0
MOVL C00004 V=800.0 PL=0
MOVL C00005 V=800.0 PL=0
MOVL C00006 V=800.0 PL=0
MOVL C00007 V=800.0 PL=0
MOVL C00008 V=800.0 PL=0
MOVL C00009 V=800.0 PL=0
MOVL C00010 V=800.0 PL=0
MOVL C00011 V=800.0 PL=0
MOVL C00012 V=800.0 PL=0
MOVL C00013 V=800.0 PL=0
MOVL C00014 V=800.0 PL=0
MOVL C00015 V=800.0 PL=0
MOVL C00016 V=800.0 PL=0
MOVL C00017 V=800.0 PL=0
MOVL C00018 V=800.0 PL=0
MOVL C00019 V=800.0 PL=0
MOVL C00020 V=800.0 PL=0
MOVL C00021 V=800.0 PL=0
MOVL C00022 V=800.0 PL=0
MOVL C00023 V=800.0 PL=0
MOVL C00024 V=800.0 PL=0
MOVL C00025 V=800.0 PL=0
MOVL C00026 V=800.0 PL=0
MOVL C00027 V=800.0 PL=0
MOVL C00028 V=800.0 PL=0
MOVL C00029 V=800.0 PL=0
MOVL C00030 V=800.0 PL=0
MOVL C00031 V=800.0 PL=0
MOVL C00032 V=800.0 PL=0
MOVL C00033 V=800.0 PL=0
MOVL C00034 V=800.0 PL=0
MOVL C00035 V=800.0 PL=0
MOVL C00036 V=800.0 PL=0
MOVL C00037 V=800.0 PL=0
MOVL C00038 V=800.0 PL=0
MOVL C00039 V=800.0 PL=0
MOVL C00040 V=800.0 PL=0
MOVL C00041 V=800.0 PL=0
MOVL C00042 V=800.0 PL=0
MOVL C00043 V=800.0 PL=0
MOVL C00044 V=800.0 PL=0
MOVL C00045 V=800.0 PL=0
MOVL C00046 V=800.0 PL=0
MOVL C00047 V=800.0 PL=0
MOVL C00048 V=800.0 PL=0
MOVL C00049 V=800.0 PL=0
MOVL C00050 V=800.0 PL=0
MOVL C00051 V=800.0 PL=0
MOVL C00052 V=800.0 PL=0
MOVL C00053 V=800.0 PL=0
MOVL C00054 V=800.0 PL=0
MOVL C00055 V=800.0 PL=0
MOVL C00056 V=800.0 PL=0
MOVL C00057 V=800.0 PL=0
MOVL C00058 V=800.0 PL=0
MOVL C00059 V=800.0 PL=0
MOVL C00060 V=800.0 PL=0
MOVL C00061 V=800.0 PL=0
MOVL C00062 V=800.0 PL=0
MOVL C00063 V=800.0 PL=0
MOVL C00064 V=800.0 PL=0
MOVL C00065 V=800.0 PL=0
MOVL C00066 V=800.0 PL=0
MOVL C00067 V=800.0 PL=0
MOVL C00068 V=800.0 PL=0
MOVL C00069 V=800.0 PL=0
MOVL C00070 V=800.0 PL=0
MOVL C00071 V=800.0 PL=0
MOVL C00072 V=800.0 PL=0
MOVL C00073 V=800.0 PL=0
MOVL C00074 V=800.0 PL=0
MOVL C00075 V=800.0 PL=0
MOVL C00076 V=800.0 PL=0
MOVL C00077 V=800.0 PL=0
MOVL C00078 V=800.0 PL=0
MOVL C00079 V=800.0 PL=0
MOVL C00080 V=800.0 PL=0
MOVL C00081 V=800.0 PL=0
MOVL C00082 V=800.0 PL=0
MOVL C00083 V=800.0 PL=0
MOVL C00084 V=800.0 PL=0
MOVL C00085 V=800.0 PL=0
MOVL C00086 V=800.0 PL=0
MOVL C00087 V=800.0 PL=0
MOVL C00088 V=800.0 PL=0
MOVL C00089 V=800.0 PL=0
MOVL C00090 V=800.0 PL=0
MOVL C00091 V=800.0 PL=0
MOVL C00092 V=800.0 PL=0
MOVL C00093 V=800.0 PL=0
MOVL C00094 V=800.0 PL=0
MOVL C00095 V=800.0 PL=0
MOVL C00096 V=800.0 PL=0
MOVL C00097 V=800.0 PL=0
MOVL C00098 V=800.0 PL=0
MOVL C00099 V=800.0 PL=0
MOVL C00100 V=800.0 PL=0
MOVL C00101 V=800.0 PL=0
MOVL C00102 V=800.0 PL=0
MOVL C00103 V=800.0 PL=0
MOVL C00104 V=800.0 PL=0
MOVL C00105 V=800.0 PL=0
MOVL C00106 V=800.0 PL=0
MOVL C00107 V=800.0 PL=0
MOVL C00108 V=800.0 PL=0
MOVL C00109 V=800.0 PL=0
MOVL C00110 V=800.0 PL=0
MOVL C00111 V=800.0 PL=0
MOVL C00112 V=800.0 PL=0
MOVL C00113 V=800.0 PL=0
MOVL C00114 V=800.0 PL=0
MOVL C00115 V=800.0 PL=0
MOVL C00116 V=800.0 PL=0
MOVL C00117 V=800.0 PL=0
MOVL C00118 V=800.0 PL=0
MOVL C00119 V=800.0 PL=0
MOVL C00120 V=800.0 PL=0
MOVL C00121 V=800.0 PL=0
MOVL C00122 V=800.0 PL=0
MOVL C00123 V=800.0 PL=0
MOVL C00124 V=800.0 PL=0
MOVL C00125 V=800.0 PL=0
MOVL C00126 V=800.0 PL=0
MOVL C00127 V=800.0 PL=0
MOVL C00128 V=800.0 PL=0
MOVL C00129 V=800.0 PL=0
MOVL C00130 V=800.0 PL=0
MOVL C00131 V=800.0 PL=0
MOVL C00132 V=800.0 PL=0
MOVL C00133 V=800.0 PL=0
MOVL C00134 V=800.0 PL=0
MOVL C00135 V=800.0 PL=0
MOVL C00136 V=800.0 PL=0
MOVL C00137 V=800.0 PL=0
MOVL C00138 V=800.0 PL=0
MOVL C00139 V=800.0 PL=0
MOVL C00140 V=800.0 PL=0
MOVL C00141 V=800.0 PL=0
MOVL C00142 V=800.0 PL=0
MOVL C00143 V=800.0 PL=0
MOVL C00144 V=800.0 PL=0
MOVL C00145 V=800.0 PL=0
MOVL C00146 V=800.0 PL=0
MOVL C00147 V=800.0 PL=0
MOVL C00148 V=800.0 PL=0
MOVL C00149 V=800.0 PL=0
MOVL C00150 V=800.0 PL=0
MOVL C00151 V=800.0 PL=0
MOVL C00152 V=800.0 PL=0
MOVL C00153 V=800.0 PL=0
MOVL C00154 V=800.0 PL=0
MOVL C00155 V=800.0 PL=0
MOVL C00156 V=800.0 PL=0
MOVL C00157 V=800.0 PL=0
MOVL C00158 V=800.0 PL=0
MOVL C00159 V=800.0 PL=0
MOVL C00160 V=800.0 PL=0
MOVL C00161 V=800.0 PL=0
MOVL C00162 V=800.0 PL=0
MOVL C00163 V=800.0 PL=0
MOVL C00164 V=800.0 PL=0
MOVL C00165 V=800.0 PL=0
MOVL C00166 V=800.0 PL=0
MOVL C00167 V=800.0 PL=0
MOVL C00168 V=800.0 PL=0
MOVL C00169 V=800.0 PL=0
MOVL C00170 V=800.0 PL=0
MOVL C00171 V=800.0 PL=0
MOVL C00172 V=800.0 PL=0
MOVL C00173 V=800.0 PL=0
MOVL C00174 V=800.0 PL=0
MOVL C00175 V=800.0 PL=0
MOVL C00176 V=800.0 PL=0
MOVL C00177 V=800.0 PL=0
MOVL C00178 V=800.0 PL=0
MOVL C00179 V=800.0 PL=0
MOVL C00180 V=800.0 PL=0
MOVL C00181 V=800.0 PL=0
MOVL C00182 V=800.0 PL=0
MOVL C00183 V=800.0 PL=0
MOVL C00184 V=800.0 PL=0
MOVL C00185 V=800.0 PL=0
MOVL C00186 V=800.0 PL=0
MOVL C00187 V=800.0 PL=0
MOVL C00188 V=800.0 PL=0
MOVL C00189 V=800.0 PL=0
MOVL C00190 V=800.0 PL=0
MOVL C00191 V=800.0 PL=0
MOVL C00192 V=800.0 PL=0
MOVL C00193 V=800.0 PL=0
MOVL C00194 V=800.0 PL=0
MOVL C00195 V=800.0 PL=0
MOVL C00196 V=800.0 PL=0
MOVL C00197 V=800.0 PL=0
MOVL C00198 V=800.0 PL=0
MOVL C00199 V=800.0 PL=0
MOVL C00200 V=800.0 PL=0
MOVL C00201 V=800.0 PL=0
MOVL C00202 V=800.0 PL=0
MOVL C00203 V=800.0 PL=0
MOVL C00204 V=800.0 PL=0
MOVL C00205 V=800.0 PL=0
MOVL C00206 V=800.0 PL=0
MOVL C00207 V=800.0 PL=0
MOVL C00208 V=800.0 PL=0
MOVL C00209 V=800.0 PL=0
MOVL C00210 V=800.0 PL=0
MOVL C00211 V=800.0 PL=0
MOVL C00212 V=800.0 PL=0
MOVL C00213 V=800.0 PL=0
MOVL C00214 V=800.0 PL=0
MOVL C00215 V=800.0 PL=0
MOVL C00216 V=800.0 PL=0
MOVL C00217 V=800.0 PL=0
MOVL C00218 V=800.0 PL=0
MOVL C00219 V=800.0 PL=0
MOVL C00220 V=800.0 PL=0
MOVL C00221 V=800.0 PL=0
MOVL C00222 V=800.0 PL=0
MOVL C00223 V=800.0 PL=0
MOVL C00224 V=800.0 PL=0
MOVL C00225 V=800.0 PL=0
MOVL C00226 V=800.0 PL=0
MOVL C00227 V=800.0 PL=0
MOVL C00228 V=800.0 PL=0
MOVL C00229 V=800.0 PL=0
MOVL C00230 V=800.0 PL=0
MOVL C00231 V=800.0 PL=0
MOVL C00232 V=800.0 PL=0
MOVL C00233 V=800.0 PL=0
MOVL C00234 V=800.0 PL=0
MOVL C00235 V=800.0 PL=0
MOVL C00236 V=800.0 PL=0
MOVL C00237 V=800.0 PL=0
MOVL C00238 V=800.0 PL=0
MOVL C00239 V=800.0 PL=0
MOVL C00240 V=800.0 PL=0
MOVL C00241 V=800.0 PL=0
MOVL C00242 V=800.0 PL=0
MOVL C00243 V=800.0 PL=0
MOVL C00244 V=800.0 PL=0
MOVL C00245 V=800.0 PL=0
MOVL C00246 V=800.0 PL=0
MOVL C00247 V=800.0 PL=0
MOVL C00248 V=800.0 PL=0
MOVL C00249 V=800.0 PL=0
MOVL C00250 V=800.0 PL=0
MOVL C00251 V=800.0 PL=0
MOVL C00252 V=800.0 PL=0
MOVL C00253 V=800.0 PL=0
MOVL C00254 V=800.0 PL=0
MOVL C00255 V=800.0 PL=0
MOVL C00256 V=800.0 PL=0
MOVL C00257 V=800.0 PL=0
MOVL C00258 V=800.0 PL=0
MOVL C00259 V=800.0 PL=0
MOVL C00260 V=800.0 PL=0
MOVL C00261 V=800.0 PL=0
MOVL C00262 V=800.0 PL=0
MOVL C00263 V=800.0 PL=0
MOVL C00264 V=800.0 PL=0
MOVL C00265 V=800.0 PL=0
MOVL C00266 V=800.0 PL=0
MOVL C00267 V=800.0 PL=0
MOVL C00268 V=800.0 PL=0
MOVL C00269 V=800.0 PL=0
MOVL C00270 V=800.0 PL=0
MOVL C00271 V=800.0 PL=0
MOVL C00272 V=800.0 PL=0
MOVL C00273 V=800.0 PL=0
MOVL C00274 V=800.0 PL=0
MOVL C00275 V=800.0 PL=0
MOVL C00276 V=800.0 PL=0
MOVL C00277 V=800.0 PL=0
MOVL C00278 V=800.0 PL=0
MOVL C00279 V=800.0 PL=0
MOVL C00280 V=800.0 PL=0
MOVL C00281 V=800.0 PL=0
MOVL C00282 V=800.0 PL=0
MOVL C00283 V=800.0 PL=0
MOVL C00284 V=800.0 PL=0
MOVL C00285 V=800.0 PL=0
MOVL C00286 V=800.0 PL=0
MOVL C00287 V=800.0 PL=0
MOVL C00288 V=800.0 PL=0
MOVL C00289 V=800.0 PL=0
MOVL C00290 V=800.0 PL=0
MOVL C00291 V=800.0 PL=0
MOVL C00292 V=800.0 PL=0
MOVL C00293 V=800.0 PL=0
MOVL C00294 V=800.0 PL=0
MOVL C00295 V=800.0 PL=0
MOVL C00296 V=800.0 PL=0
MOVL C00297 V=800.0 PL=0
MOVL C00298 V=800.0 PL=0
MOVL C00299 V=800.0 PL=0
MOVL C00300 V=800.0 PL=0
MOVL C00301 V=800.0 PL=0
MOVL C00302 V=800.0 PL=0
MOVL C00303 V=800.0 PL=0
MOVL C00304 V=800.0 PL=0
MOVL C00305 V=800.0 PL=0
MOVL C00306 V=800.0 PL=0
MOVL C00307 V=800.0 PL=0
MOVL C00308 V=800.0 PL=0
MOVL C00309 V=800.0 PL=0
MOVL C00310 V=800.0 PL=0
MOVL C00311 V=800.0 PL=0
MOVL C00312 V=800.0 PL=0
MOVL C00313 V=800.0 PL=0
MOVL C00314 V=800.0 PL=0
MOVL C00315 V=800.0 PL=0
MOVL C00316 V=800.0 PL=0
MOVL C00317 V=800.0 PL=0
MOVL C00318 V=800.0 PL=0
MOVL C00319 V=800.0 PL=0
MOVL C00320 V=800.0 PL=0
MOVL C00321 V=800.0 PL=0
MOVL C00322 V=800.0 PL=0
MOVL C00323 V=800.0 PL=0
MOVL C00324 V=800.0 PL=0
MOVL C00325 V=800.0 PL=0
MOVL C00326 V=800.0 PL=0
MOVL C00327 V=800.0 PL=0
MOVL C00328 V=800.0 PL=0
MOVL C00329 V=800.0 PL=0
MOVL C00330 V=800.0 PL=0
MOVL C00331 V=800.0 PL=0
MOVL C00332 V=800.0 PL=0
MOVL C00333 V=800.0 PL=0
MOVL C00334 V=800.0 PL=0
MOVL C00335 V=800.0 PL=0
MOVL C00336 V=800.0 PL=0
MOVL C00337 V=800.0 PL=0
MOVL C00338 V=800.0 PL=0
MOVL C00339 V=800.0 PL=0
MOVL C00340 V=800.0 PL=0
MOVL C00341 V=800.0 PL=0
MOVL C00342 V=800.0 PL=0
MOVL C00343 V=800.0 PL=0
MOVL C00344 V=800.0 PL=0
MOVL C00345 V=800.0 PL=0
MOVL C00346 V=800.0 PL=0
MOVL C00347 V=800.0 PL=0
MOVL C00348 V=800.0 PL=0
MOVL C00349 V=800.0 PL=0
MOVL C00350 V=800.0 PL=0
MOVL C00351 V=800.0 PL=0
MOVL C00352 V=800.0 PL=0
MOVL C00353 V=800.0 PL=0
MOVL C00354 V=800.0 PL=0
MOVL C00355 V=800.0 PL=0
MOVL C00356 V=800.0 PL=0
MOVL C00357 V=800.0 PL=0
MOVL C00358 V=800.0 PL=0
MOVL C00359 V=800.0 PL=0
MOVL C00360 V=800.0 PL=0
MOVL C00361 V=800.0 PL=0
MOVL C00362 V=800.0 PL=0
MOVL C00363 V=800.0 PL=0
MOVL C00364 V=800.0 PL=0
MOVL C00365 V=800.0 PL=0
MOVL C00366 V=800.0 PL=0
MOVL C00367 V=800.0 PL=0
MOVL C00368 V=800.0 PL=0
MOVL C00369 V=800.0 PL=0
MOVL C00370 V=800.0 PL=0
MOVL C00371 V=800.0 PL=0
MOVL C00372 V=800.0 PL=0
MOVL C00373 V=800.0 PL=0
MOVL C00374 V=800.0 PL=0
MOVL C00375 V=800.0 PL=0
MOVL C00376 V=800.0 PL=0
MOVL C00377 V=800.0 PL=0
MOVL C00378 V=800.0 PL=0
MOVL C00379 V=800.0 PL=0
MOVL C00380 V=800.0 PL=0
MOVL C00381 V=800.0 PL=0
MOVL C00382 V=800.0 PL=0
MOVL C00383 V=800.0 PL=0
MOVL C00384 V=800.0 PL=0
MOVL C00385 V=800.0 PL=0
MOVL C00386 V=800.0 PL=0
MOVL C00387 V=800.0 PL=0
MOVL C00388 V=800.0 PL=0
MOVL C00389 V=800.0 PL=0
MOVL C00390 V=800.0 PL=0
MOVL C00391 V=800.0 PL=0
MOVL C00392 V=800.0 PL=0
MOVL C00393 V=800.0 PL=0
MOVL C00394 V=800.0 PL=0
MOVL C00395 V=800.0 PL=0
MOVL C00396 V=800.0 PL=0
MOVL C00397 V=800.0 PL=0
MOVL C00398 V=800.0 PL=0
MOVL C00399 V=800.0 PL=0
MOVL C00400 V=800.0 PL=0
MOVL C00401 V=800.0 PL=0
MOVL C00402 V=800.0 PL=0
MOVL C00403 V=800.0 PL=0
MOVL C00404 V=800.0 PL=0
MOVL C00405 V=800.0 PL=0
MOVL C00406 V=800.0 PL=0
MOVL C00407 V=800.0 PL=0
MOVL C00408 V=800.0 PL=0
MOVL C00409 V=800.0 PL=0
MOVL C00410 V=800.0 PL=0
MOVL C00411 V=800.0 PL=0
MOVL C00412 V=800.0 PL=0
MOVL C00413 V=800.0 PL=0
MOVL C00414 V=800.0 PL=0
MOVL C00415 V=800.0 PL=0
MOVL C00416 V=800.0 PL=0
MOVL C00417 V=800.0 PL=0
MOVL C00418 V=800.0 PL=0
MOVL C00419 V=800.0 PL=0
MOVL C00420 V=800.0 PL=0
MOVL C00421 V=800.0 PL=0
MOVL C00422 V=800.0 PL=0
MOVL C00423 V=800.0 PL=0
MOVL C00424 V=800.0 PL=0
MOVL C00425 V=800.0 PL=0
MOVL C00426 V=800.0 PL=0
MOVL C00427 V=800.0 PL=0
MOVL C00428 V=800.0 PL=0
MOVL C00429 V=800.0 PL=0
MOVL C00430 V=800.0 PL=0
MOVL C00431 V=800.0 PL=0
MOVL C00432 V=800.0 PL=0
MOVL C00433 V=800.0 PL=0
MOVL C00434 V=800.0 PL=0
MOVL C00435 V=800.0 PL=0
MOVL C00436 V=800.0 PL=0
MOVL C00437 V=800.0 PL=0
MOVL C00438 V=800.0 PL=0
MOVL C00439 V=800.0 PL=0
MOVL C00440 V=800.0 PL=0
MOVL C00441 V=800.0 PL=0
MOVL C00442 V=800.0 PL=0
MOVL C00443 V=800.0 PL=0
MOVL C00444 V=800.0 PL=0
MOVL C00445 V=800.0 PL=0
MOVL C00446 V=800.0 PL=0
MOVL C00447 V=800.0 PL=0
MOVL C00448 V=800.0 PL=0
MOVL C00449 V=800.0 PL=0
MOVL C00450 V=800.0 PL=0
MOVL C00451 V=800.0 PL=0
MOVL C00452 V=800.0 PL=0
MOVL C00453 V=800.0 PL=0
MOVL C00454 V=800.0 PL=0
MOVL C00455 V=800.0 PL=0
MOVL C00456 V=800.0 PL=0
MOVL C00457 V=800.0 PL=0
MOVL C00458 V=800.0 PL=0
MOVL C00459 V=800.0 PL=0
MOVL C00460 V=800.0 PL=0
MOVL C00461 V=800.0 PL=0
MOVL C00462 V=800.0 PL=0
MOVL C00463 V=800.0 PL=0
MOVL C00464 V=800.0 PL=0
MOVL C00465 V=800.0 PL=0
MOVL C00466 V=800.0 PL=0
MOVL C00467 V=800.0 PL=0
MOVL C00468 V=800.0 PL=0
MOVL C00469 V=800.0 PL=0
MOVL C00470 V=800.0 PL=0
MOVL C00471 V=800.0 PL=0
MOVL C00472 V=800.0 PL=0
MOVL C00473 V=800.0 PL=0
MOVL C00474 V=800.0 PL=0
MOVL C00475 V=800.0 PL=0
MOVL C00476 V=800.0 PL=0
MOVL C00477 V=800.0 PL=0
MOVL C00478 V=800.0 PL=0
MOVL C00479 V=800.0 PL=0
MOVL C00480 V=800.0 PL=0
MOVL C00481 V=800.0 PL=0
MOVL C00482 V=800.0 PL=0
MOVL C00483 V=800.0 PL=0
MOVL C00484 V=800.0 PL=0
MOVL C00485 V=800.0 PL=0
MOVL C00486 V=800.0 PL=0
MOVL C00487 V=800.0 PL=0
MOVL C00488 V=800.0 PL=0
MOVL C00489 V=800.0 PL=0
MOVL C00490 V=800.0 PL=0
MOVL C00491 V=800.0 PL=0
MOVL C00492 V=800.0 PL=0
MOVL C00493 V=800.0 PL=0
MOVL C00494 V=800.0 PL=0
MOVL C00495 V=800.0 PL=0
MOVL C00496 V=800.0 PL=0
MOVL C00497 V=800.0 PL=0
MOVL C00498 V=800.0 PL=0
MOVL C00499 V=800.0 PL=0
MOVL C00500 V=800.0 PL=0
MOVL C00501 V=800.0 PL=0
MOVL C00502 V=800.0 PL=0
MOVL C00503 V=800.0 PL=0
MOVL C00504 V=800.0 PL=0
MOVL C00505 V=800.0 PL=0
MOVL C00506 V=800.0 PL=0
MOVL C00507 V=800.0 PL=0
MOVL C00508 V=800.0 PL=0
MOVL C00509 V=800.0 PL=0
MOVL C00510 V=800.0 PL=0
MOVL C00511 V=800.0 PL=0
MOVL C00512 V=800.0 PL=0
MOVL C00513 V=800.0 PL=0
MOVL C00514 V=800.0 PL=0
MOVL C00515 V=800.0 PL=0
MOVL C00516 V=800.0 PL=0
MOVL C00517 V=800.0 PL=0
MOVL C00518 V=800.0 PL=0
MOVL C00519 V=800.0 PL=0
MOVL C00520 V=800.0 PL=0
MOVL C00521 V=800.0 PL=0
MOVL C00522 V=800.0 PL=0
MOVL C00523 V=800.0 PL=0
MOVL C00524 V=800.0 PL=0
MOVL C00525 V=800.0 PL=0
MOVL C00526 V=800.0 PL=0
MOVL C00527 V=800.0 PL=0
MOVL C00528 V=800.0 PL=0
MOVL C00529 V=800.0 PL=0
MOVL C00530 V=800.0 PL=0
MOVL C00531 V=800.0 PL=0
MOVL C00532 V=800.0 PL=0
MOVL C00533 V=800.0 PL=0
MOVL C00534 V=800.0 PL=0
MOVL C00535 V=800.0 PL=0
MOVL C00536 V=800.0 PL=0
MOVL C00537 V=800.0 PL=0
MOVL C00538 V=800.0 PL=0
MOVL C00539 V=800.0 PL=0
MOVL C00540 V=800.0 PL=0
MOVL C00541 V=800.0 PL=0
MOVL C00542 V=800.0 PL=0
MOVL C00543 V=800.0 PL=0
MOVL C00544 V=800.0 PL=0
MOVL C00545 V=800.0 PL=0
MOVL C00546 V=800.0 PL=0
MOVL C00547 V=800.0 PL=0
MOVL C00548 V=800.0 PL=0
MOVL C00549 V=800.0 PL=0
MOVL C00550 V=800.0 PL=0
MOVL C00551 V=800.0 PL=0
MOVL C00552 V=800.0 PL=0
MOVL C00553 V=800.0 PL=0
MOVL C00554 V=800.0 PL=0
MOVL C00555 V=800.0 PL=0
MOVL C00556 V=800.0 PL=0
MOVL C00557 V=800.0 PL=0
MOVL C00558 V=800.0 PL=0
MOVL C00559 V=800.0 PL=0
MOVL C00560 V=800.0 PL=0
MOVL C00561 V=800.0 PL=0
MOVL C00562 V=800.0 PL=0
MOVL C00563 V=800.0 PL=0
MOVL C00564 V=800.0 PL=0
MOVL C00565 V=800.0 PL=0
MOVL C00566 V=800.0 PL=0
MOVL C00567 V=800.0 PL=0
MOVL C00568 V=800.0 PL=0
MOVL C00569 V=800.0 PL=0
MOVL C00570 V=800.0 PL=0
MOVL C00571 V=800.0 PL=0
MOVL C00572 V=800.0 PL=0
MOVL C00573 V=800.0 PL=0
MOVL C00574 V=800.0 PL=0
MOVL C00575 V=800.0 PL=0
MOVL C00576 V=800.0 PL=0
MOVL C00577 V=800.0 PL=0
MOVL C00578 V=800.0 PL=0
MOVL C00579 V=800.0 PL=0
MOVL C00580 V=800.0 PL=0
MOVL C00581 V=800.0 PL=0
MOVL C00582 V=800.0 PL=0
MOVL C00583 V=800.0 PL=0
MOVL C00584 V=800.0 PL=0
MOVL C00585 V=800.0 PL=0
MOVL C00586 V=800.0 PL=0
MOVL C00587 V=800.0 PL=0
MOVL C00588 V=800.0 PL=0
MOVL C00589 V=800.0 PL=0
MOVL C00590 V=800.0 PL=0
MOVL C00591 V=800.0 PL=0
MOVL C00592 V=800.0 PL=0
MOVL C00593 V=800.0 PL=0
MOVL C00594 V=800.0 PL=0
MOVL C00595 V=800.0 PL=0
MOVL C00596 V=800.0 PL=0
MOVL C00597 V=800.0 PL=0
MOVL C00598 V=800.0 PL=0
MOVL C00599 V=800.0 PL=0
MOVL C00600 V=800.0 PL=0
MOVL C00601 V=800.0 PL=0
MOVL C00602 V=800.0 PL=0
MOVL C00603 V=800.0 PL=0
MOVL C00604 V=800.0 PL=0
MOVL C00605 V=800.0 PL=0
MOVL C00606 V=800.0 PL=0
MOVL C00607 V=800.0 PL=0
MOVL C00608 V=800.0 PL=0
MOVL C00609 V=800.0 PL=0
MOVL C00610 V=800.0 PL=0
MOVL C00611 V=800.0 PL=0
MOVL C00612 V=800.0 PL=0
MOVL C00613 V=800.0 PL=0
MOVL C00614 V=800.0 PL=0
MOVL C00615 V=800.0 PL=0
MOVL C00616 V=800.0 PL=0
MOVL C00617 V=800.0 PL=0
MOVL C00618 V=800.0 PL=0
MOVL C00619 V=800.0 PL=0
MOVL C00620 V=800.0 PL=0
MOVL C00621 V=800.0 PL=0
MOVL C00622 V=800.0 PL=0
MOVL C00623 V=800.0 PL=0
MOVL C00624 V=800.0 PL=0
MOVL C00625 V=800.0 PL=0
MOVL C00626 V=800.0 PL=0
MOVL C00627 V=800.0 PL=0
MOVL C00628 V=800.0 PL=0
MOVL C00629 V=800.0 PL=0
MOVL C00630 V=800.0 PL=0
MOVL C00631 V=800.0 PL=0
MOVL C00632 V=800.0 PL=0
MOVL C00633 V=800.0 PL=0
MOVL C00634 V=800.0 PL=0
MOVL C00635 V=800.0 PL=0
MOVL C00636 V=800.0 PL=0
MOVL C00637 V=800.0 PL=0
MOVL C00638 V=800.0 PL=0
MOVL C00639 V=800.0 PL=0
MOVL C00640 V=800.0 PL=0
MOVL C00641 V=800.0 PL=0
MOVL C00642 V=800.0 PL=0
MOVL C00643 V=800.0 PL=0
MOVL C00644 V=800.0 PL=0
MOVL C00645 V=800.0 PL=0
MOVL C00646 V=800.0 PL=0
MOVL C00647 V=800.0 PL=0
MOVL C00648 V=800.0 PL=0
MOVL C00649 V=800.0 PL=0
MOVL C00650 V=800.0 PL=0
MOVL C00651 V=800.0 PL=0
MOVL C00652 V=800.0 PL=0
MOVL C00653 V=800.0 PL=0
MOVL C00654 V=800.0 PL=0
MOVL C00655 V=800.0 PL=0
MOVL C00656 V=800.0 PL=0
MOVL C00657 V=800.0 PL=0
MOVL C00658 V=800.0 PL=0
MOVL C00659 V=800.0 PL=0
MOVL C00660 V=800.0 PL=0
MOVL C00661 V=800.0 PL=0
MOVL C00662 V=800.0 PL=0
MOVL C00663 V=800.0 PL=0
MOVL C00664 V=800.0 PL=0
MOVL C00665 V=800.0 PL=0
MOVL C00666 V=800.0 PL=0
MOVL C00667 V=800.0 PL=0
MOVL C00668 V=800.0 PL=0
MOVL C00669 V=800.0 PL=0
MOVL C00670 V=800.0 PL=0
MOVL C00671 V=800.0 PL=0
MOVL C00672 V=800.0 PL=0
MOVL C00673 V=800.0 PL=0
MOVL C00674 V=800.0 PL=0
MOVL C00675 V=800.0 PL=0
MOVL C00676 V=800.0 PL=0
MOVL C00677 V=800.0 PL=0
MOVL C00678 V=800.0 PL=0
MOVL C00679 V=800.0 PL=0
MOVL C00680 V=800.0 PL=0
MOVL C00681 V=800.0 PL=0
MOVL C00682 V=800.0 PL=0
MOVL C00683 V=800.0 PL=0
MOVL C00684 V=800.0 PL=0
MOVL C00685 V=800.0 PL=0
MOVL C00686 V=800.0 PL=0
MOVL C00687 V=800.0 PL=0
MOVL C00688 V=800.0 PL=0
MOVL C00689 V=800.0 PL=0
MOVL C00690 V=800.0 PL=0
MOVL C00691 V=800.0 PL=0
MOVL C00692 V=800.0 PL=0
MOVL C00693 V=800.0 PL=0
MOVL C00694 V=800.0 PL=0
MOVL C00695 V=800.0 PL=0
MOVL C00696 V=800.0 PL=0
MOVL C00697 V=800.0 PL=0
MOVL C00698 V=800.0 PL=0
MOVL C00699 V=800.0 PL=0
MOVL C00700 V=800.0 PL=0
MOVL C00701 V=800.0 PL=0
MOVL C00702 V=800.0 PL=0
MOVL C00703 V=800.0 PL=0
MOVL C00704 V=800.0 PL=0
MOVL C00705 V=800.0 PL=0
MOVL C00706 V=800.0 PL=0
MOVL C00707 V=800.0 PL=0
MOVL C00708 V=800.0 PL=0
MOVL C00709 V=800.0 PL=0
MOVL C00710 V=800.0 PL=0
MOVL C00711 V=800.0 PL=0
MOVL C00712 V=800.0 PL=0
MOVL C00713 V=800.0 PL=0
MOVL C00714 V=800.0 PL=0
MOVL C00715 V=800.0 PL=0
MOVL C00716 V=800.0 PL=0
MOVL C00717 V=800.0 PL=0
MOVL C00718 V=800.0 PL=0
MOVL C00719 V=800.0 PL=0
MOVL C00720 V=800.0 PL=0
MOVL C00721 V=800.0 PL=0
MOVL C00722 V=800.0 PL=0
MOVL C00723 V=800.0 PL=0
MOVL C00724 V=800.0 PL=0
MOVL C00725 V=800.0 PL=0
MOVL C00726 V=800.0 PL=0
MOVL C00727 V=800.0 PL=0
MOVL C00728 V=800.0 PL=0
MOVL C00729 V=800.0 PL=0
MOVL C00730 V=800.0 PL=0
MOVL C00731 V=800.0 PL=0
MOVL C00732 V=800.0 PL=0
MOVL C00733 V=800.0 PL=0
MOVL C00734 V=800.0 PL=0
MOVL C00735 V=800.0 PL=0
MOVL C00736 V=800.0 PL=0
MOVL C00737 V=800.0 PL=0
MOVL C00738 V=800.0 PL=0
MOVL C00739 V=800.0 PL=0
MOVL C00740 V=800.0 PL=0
MOVL C00741 V=800.0 PL=0
MOVL C00742 V=800.0 PL=0
MOVL C00743 V=800.0 PL=0
MOVL C00744 V=800.0 PL=0
MOVL C00745 V=800.0 PL=0
MOVL C00746 V=800.0 PL=0
MOVL C00747 V=800.0 PL=0
MOVL C00748 V=800.0 PL=0
MOVL C00749 V=800.0 PL=0
MOVL C00750 V=800.0 PL=0
MOVL C00751 V=800.0 PL=0
MOVL C00752 V=800.0 PL=0
MOVL C00753 V=800.0 PL=0
MOVL C00754 V=800.0 PL=0
MOVL C00755 V=800.0 PL=0
MOVL C00756 V=800.0 PL=0
MOVL C00757 V=800.0 PL=0
MOVL C00758 V=800.0 PL=0
MOVL C00759 V=800.0 PL=0
MOVL C00760 V=800.0 PL=0
MOVL C00761 V=800.0 PL=0
MOVL C00762 V=800.0 PL=0
MOVL C00763 V=800.0 PL=0
MOVL C00764 V=800.0 PL=0
MOVL C00765 V=800.0 PL=0
MOVL C00766 V=800.0 PL=0
MOVL C00767 V=800.0 PL=0
MOVL C00768 V=800.0 PL=0
MOVL C00769 V=800.0 PL=0
MOVL C00770 V=800.0 PL=0
MOVL C00771 V=800.0 PL=0
MOVL C00772 V=800.0 PL=0
MOVL C00773 V=800.0 PL=0
MOVL C00774 V=800.0 PL=0
MOVL C00775 V=800.0 PL=0
MOVL C00776 V=800.0 PL=0
MOVL C00777 V=800.0 PL=0
MOVL C00778 V=800.0 PL=0
MOVL C00779 V=800.0 PL=0
MOVL C00780 V=800.0 PL=0
MOVL C00781 V=800.0 PL=0
MOVL C00782 V=800.0 PL=0
MOVL C00783 V=800.0 PL=0
MOVL C00784 V=800.0 PL=0
MOVL C00785 V=800.0 PL=0
MOVL C00786 V=800.0 PL=0
MOVL C00787 V=800.0 PL=0
MOVL C00788 V=800.0 PL=0
MOVL C00789 V=800.0 PL=0
MOVL C00790 V=800.0 PL=0
MOVL C00791 V=800.0 PL=0
MOVL C00792 V=800.0 PL=0
MOVL C00793 V=800.0 PL=0
MOVL C00794 V=800.0 PL=0
MOVL C00795 V=800.0 PL=0
MOVL C00796 V=800.0 PL=0
MOVL C00797 V=800.0 PL=0
MOVL C00798 V=800.0 PL=0
MOVL C00799 V=800.0 PL=0
MOVL C00800 V=800.0 PL=0
MOVL C00801 V=800.0 PL=0
MOVL C00802 V=800.0 PL=0
MOVL C00803 V=800.0 PL=0
MOVL C00804 V=800.0 PL=0
MOVL C00805 V=800.0 PL=0
MOVL C00806 V=800.0 PL=0
MOVL C00807 V=800.0 PL=0
MOVL C00808 V=800.0 PL=0
MOVL C00809 V=800.0 PL=0
MOVL C00810 V=800.0 PL=0
MOVL C00811 V=800.0 PL=0
MOVL C00812 V=800.0 PL=0
MOVL C00813 V=800.0 PL=0
MOVL C00814 V=800.0 PL=0
MOVL C00815 V=800.0 PL=0
MOVL C00816 V=800.0 PL=0
MOVL C00817 V=800.0 PL=0
MOVL C00818 V=800.0 PL=0
MOVL C00819 V=800.0 PL=0
MOVL C00820 V=800.0 PL=0
MOVL C00821 V=800.0 PL=0
MOVL C00822 V=800.0 PL=0
MOVL C00823 V=800.0 PL=0
MOVL C00824 V=800.0 PL=0
MOVL C00825 V=800.0 PL=0
MOVL C00826 V=800.0 PL=0
MOVL C00827 V=800.0 PL=0
MOVL C00828 V=800.0 PL=0
MOVL C00829 V=800.0 PL=0
MOVL C00830 V=800.0 PL=0
MOVL C00831 V=800.0 PL=0
MOVL C00832 V=800.0 PL=0
MOVL C00833 V=800.0 PL=0
MOVL C00834 V=800.0 PL=0
MOVL C00835 V=800.0 PL=0
MOVL C00836 V=800.0 PL=0
MOVL C00837 V=800.0 PL=0
MOVL C00838 V=800.0 PL=0
MOVL C00839 V=800.0 PL=0
MOVL C00840 V=800.0 PL=0
MOVL C00841 V=800.0 PL=0
MOVL C00842 V=800.0 PL=0
MOVL C00843 V=800.0 PL=0
MOVL C00844 V=800.0 PL=0
MOVL C00845 V=800.0 PL=0
MOVL C00846 V=800.0 PL=0
MOVL C00847 V=800.0 PL=0
MOVL C00848 V=800.0 PL=0
MOVL C00849 V=800.0 PL=0
MOVL C00850 V=800.0 PL=0
MOVL C00851 V=800.0 PL=0
MOVL C00852 V=800.0 PL=0
MOVL C00853 V=800.0 PL=0
MOVL C00854 V=800.0 PL=0
MOVL C00855 V=800.0 PL=0
MOVL C00856 V=800.0 PL=0
MOVL C00857 V=800.0 PL=0
MOVL C00858 V=800.0 PL=0
MOVL C00859 V=800.0 PL=0
MOVL C00860 V=800.0 PL=0
MOVL C00861 V=800.0 PL=0
MOVL C00862 V=800.0 PL=0
MOVL C00863 V=800.0 PL=0
MOVL C00864 V=800.0 PL=0
MOVL C00865 V=800.0 PL=0
MOVL C00866 V=800.0 PL=0
MOVL C00867 V=800.0 PL=0
MOVL C00868 V=800.0 PL=0
MOVL C00869 V=800.0 PL=0
MOVL C00870 V=800.0 PL=0
MOVL C00871 V=800.0 PL=0
MOVL C00872 V=800.0 PL=0
MOVL C00873 V=800.0 PL=0
MOVL C00874 V=800.0 PL=0
MOVL C00875 V=800.0 PL=0
MOVL C00876 V=800.0 PL=0
MOVL C00877 V=800.0 PL=0
MOVL C00878 V=800.0 PL=0
MOVL C00879 V=800.0 PL=0
MOVL C00880 V=800.0 PL=0
MOVL C00881 V=800.0 PL=0
MOVL C00882 V=800.0 PL=0
MOVL C00883 V=800.0 PL=0
MOVL C00884 V=800.0 PL=0
MOVL C00885 V=800.0 PL=0
MOVL C00886 V=800.0 PL=0
MOVL C00887 V=800.0 PL=0
MOVL C00888 V=800.0 PL=0
MOVL C00889 V=800.0 PL=0
MOVL C00890 V=800.0 PL=0
MOVL C00891 V=800.0 PL=0
MOVL C00892 V=800.0 PL=0
MOVL C00893 V=800.0 PL=0
MOVL C00894 V=800.0 PL=0
MOVL C00895 V=800.0 PL=0
MOVL C00896 V=800.0 PL=0
MOVL C00897 V=800.0 PL=0
MOVL C00898 V=800.0 PL=0
MOVL C00899 V=800.0 PL=0
MOVL C00900 V=800.0 PL=0
MOVL C00901 V=800.0 PL=0
MOVL C00902 V=800.0 PL=0
MOVL C00903 V=800.0 PL=0
MOVL C00904 V=800.0 PL=0
MOVL C00905 V=800.0 PL=0
MOVL C00906 V=800.0 PL=0
MOVL C00907 V=800.0 PL=0
MOVL C00908 V=800.0 PL=0
MOVL C00909 V=800.0 PL=0
MOVL C00910 V=800.0 PL=0
MOVL C00911 V=800.0 PL=0
MOVL C00912 V=800.0 PL=0
MOVL C00913 V=800.0 PL=0
MOVL C00914 V=800.0 PL=0
MOVL C00915 V=800.0 PL=0
MOVL C00916 V=800.0 PL=0
MOVL C00917 V=800.0 PL=0
MOVL C00918 V=800.0 PL=0
MOVL C00919 V=800.0 PL=0
MOVL C00920 V=800.0 PL=0
MOVL C00921 V=800.0 PL=0
MOVL C00922 V=800.0 PL=0
MOVL C00923 V=800.0 PL=0
MOVL C00924 V=800.0 PL=0
MOVL C00925 V=800.0 PL=0
MOVL C00926 V=800.0 PL=0
MOVL C00927 V=800.0 PL=0
MOVL C00928 V=800.0 PL=0
MOVL C00929 V=800.0 PL=0
MOVL C00930 V=800.0 PL=0
MOVL C00931 V=800.0 PL=0
MOVL C00932 V=800.0 PL=0
MOVL C00933 V=800.0 PL=0
MOVL C00934 V=800.0 PL=0
MOVL C00935 V=800.0 PL=0
MOVL C00936 V=800.0 PL=0
MOVL C00937 V=800.0 PL=0
MOVL C00938 V=800.0 PL=0
MOVL C00939 V=800.0 PL=0
MOVL C00940 V=800.0 PL=0
MOVL C00941 V=800.0 PL=0
MOVL C00942 V=800.0 PL=0
MOVL C00943 V=800.0 PL=0
MOVL C00944 V=800.0 PL=0
MOVL C00945 V=800.0 PL=0
MOVL C00946 V=800.0 PL=0
MOVL C00947 V=800.0 PL=0
MOVL C00948 V=800.0 PL=0
MOVL C00949 V=800.0 PL=0
MOVL C00950 V=800.0 PL=0
MOVL C00951 V=800.0 PL=0
MOVL C00952 V=800.0 PL=0
MOVL C00953 V=800.0 PL=0
MOVL C00954 V=800.0 PL=0
MOVL C00955 V=800.0 PL=0
MOVL C00956 V=800.0 PL=0
MOVL C00957 V=800.0 PL=0
MOVL C00958 V=800.0 PL=0
MOVL C00959 V=800.0 PL=0
MOVL C00960 V=800.0 PL=0
MOVL C00961 V=800.0 PL=0
MOVL C00962 V=800.0 PL=0
MOVL C00963 V=800.0 PL=0
MOVL C00964 V=800.0 PL=0
MOVL C00965 V=800.0 PL=0
MOVL C00966 V=800.0 PL=0
MOVL C00967 V=800.0 PL=0
MOVL C00968 V=800.0 PL=0
MOVL C00969 V=800.0 PL=0
MOVL C00970 V=800.0 PL=0
MOVL C00971 V=800.0 PL=0
MOVL C00972 V=800.0 PL=0
MOVL C00973 V=800.0 PL=0
MOVL C00974 V=800.0 PL=0
MOVL C00975 V=800.0 PL=0
MOVL C00976 V=800.0 PL=0
MOVL C00977 V=800.0 PL=0
MOVL C00978 V=800.0 PL=0
MOVL C00979 V=800.0 PL=0
MOVL C00980 V=800.0 PL=0
MOVL C00981 V=800.0 PL=0
MOVL C00982 V=800.0 PL=0
MOVL C00983 V=800.0 PL=0
MOVL C00984 V=800.0 PL=0
MOVL C00985 V=800.0 PL=0
MOVL C00986 V=800.0 PL=0
MOVL C00987 V=800.0 PL=0
MOVL C00988 V=800.0 PL=0
MOVL C00989 V=800.0 PL=0
MOVL C00990 V=800.0 PL=0
MOVL C00991 V=800.0 PL=0
MOVL C00992 V=800.0 PL=0
MOVL C00993 V=800.0 PL=0
MOVL C00994 V=800.0 PL=0
MOVL C00995 V=800.0 PL=0
MOVL C00996 V=800.0 PL=0
MOVL C00997 V=800.0 PL=0
MOVL C00998 V=800.0 PL=0
MOVL C00999 V=800.0 PL=0
MOVL C01000 V=800.0 PL=0
MOVL C01001 V=800.0 PL=0
MOVL C01002 V=800.0 PL=0
MOVL C01003 V=800.0 PL=0
MOVL C01004 V=800.0 PL=0
MOVL C01005 V=800.0 PL=0
MOVL C01006 V=800.0 PL=0
MOVL C01007 V=800.0 PL=0
MOVL C01008 V=800.0 PL=0
MOVL C01009 V=800.0 PL=0
MOVL C01010 V=800.0 PL=0
MOVL C01011 V=800.0 PL=0
MOVL C01012 V=800.0 PL=0
MOVL C01013 V=800.0 PL=0
MOVL C01014 V=800.0 PL=0
MOVL C01015 V=800.0 PL=0
MOVL C01016 V=800.0 PL=0
MOVL C01017 V=800.0 PL=0
MOVL C01018 V=800.0 PL=0
MOVL C01019 V=800.0 PL=0
MOVL C01020 V=800.0 PL=0
MOVL C01021 V=800.0 PL=0
MOVL C01022 V=800.0 PL=0
MOVL C01023 V=800.0 PL=0
MOVL C01024 V=800.0 PL=0
MOVL C01025 V=800.0 PL=0
MOVL C01026 V=800.0 PL=0
MOVL C01027 V=800.0 PL=0
MOVL C01028 V=800.0 PL=0
MOVL C01029 V=800.0 PL=0
MOVL C01030 V=800.0 PL=0
MOVL C01031 V=800.0 PL=0
MOVL C01032 V=800.0 PL=0
MOVL C01033 V=800.0 PL=0
MOVL C01034 V=800.0 PL=0
MOVL C01035 V=800.0 PL=0
MOVL C01036 V=800.0 PL=0
MOVL C01037 V=800.0 PL=0
MOVL C01038 V=800.0 PL=0
MOVL C01039 V=800.0 PL=0
MOVL C01040 V=800.0 PL=0
MOVL C01041 V=800.0 PL=0
MOVL C01042 V=800.0 PL=0
MOVL C01043 V=800.0 PL=0
MOVL C01044 V=800.0 PL=0
MOVL C01045 V=800.0 PL=0
MOVL C01046 V=800.0 PL=0
MOVL C01047 V=800.0 PL=0
MOVL C01048 V=800.0 PL=0
MOVL C01049 V=800.0 PL=0
MOVL C01050 V=800.0 PL=0
MOVL C01051 V=800.0 PL=0
MOVL C01052 V=800.0 PL=0
MOVL C01053 V=800.0 PL=0
MOVL C01054 V=800.0 PL=0
MOVL C01055 V=800.0 PL=0
MOVL C01056 V=800.0 PL=0
MOVL C01057 V=800.0 PL=0
MOVL C01058 V=800.0 PL=0
MOVL C01059 V=800.0 PL=0
MOVL C01060 V=800.0 PL=0
MOVL C01061 V=800.0 PL=0
MOVL C01062 V=800.0 PL=0
MOVL C01063 V=800.0 PL=0
MOVL C01064 V=800.0 PL=0
MOVL C01065 V=800.0 PL=0
MOVL C01066 V=800.0 PL=0
MOVL C01067 V=800.0 PL=0
MOVL C01068 V=800.0 PL=0
MOVL C01069 V=800.0 PL=0
MOVL C01070 V=800.0 PL=0
MOVL C01071 V=800.0 PL=0
MOVL C01072 V=800.0 PL=0
MOVL C01073 V=800.0 PL=0
MOVL C01074 V=800.0 PL=0
MOVL C01075 V=800.0 PL=0
MOVL C01076 V=800.0 PL=0
MOVL C01077 V=800.0 PL=0
MOVL C01078 V=800.0 PL=0
MOVL C01079 V=800.0 PL=0
MOVL C01080 V=800.0 PL=0
MOVL C01081 V=800.0 PL=0
MOVL C01082 V=800.0 PL=0
MOVL C01083 V=800.0 PL=0
MOVL C01084 V=800.0 PL=0
MOVL C01085 V=800.0 PL=0
MOVL C01086 V=800.0 PL=0
MOVL C01087 V=800.0 PL=0
MOVL C01088 V=800.0 PL=0
MOVL C01089 V=800.0 PL=0
MOVL C01090 V=800.0 PL=0
MOVL C01091 V=800.0 PL=0
MOVL C01092 V=800.0 PL=0
MOVL C01093 V=800.0 PL=0
MOVL C01094 V=800.0 PL=0
MOVL C01095 V=800.0 PL=0
MOVL C01096 V=800.0 PL=0
MOVL C01097 V=800.0 PL=0
MOVL C01098 V=800.0 PL=0
MOVL C01099 V=800.0 PL=0
MOVL C01100 V=800.0 PL=0
MOVL C01101 V=800.0 PL=0
MOVL C01102 V=800.0 PL=0
MOVL C01103 V=800.0 PL=0
MOVL C01104 V=800.0 PL=0
MOVL C01105 V=800.0 PL=0
MOVL C01106 V=800.0 PL=0
MOVL C01107 V=800.0 PL=0
MOVL C01108 V=800.0 PL=0
MOVL C01109 V=800.0 PL=0
MOVL C01110 V=800.0 PL=0
MOVL C01111 V=800.0 PL=0
MOVL C01112 V=800.0 PL=0
MOVL C01113 V=800.0 PL=0
MOVL C01114 V=800.0 PL=0
MOVL C01115 V=800.0 PL=0
MOVL C01116 V=800.0 PL=0
MOVL C01117 V=800.0 PL=0
MOVL C01118 V=800.0 PL=0
MOVL C01119 V=800.0 PL=0
MOVL C01120 V=800.0 PL=0
MOVL C01121 V=800.0 PL=0
MOVL C01122 V=800.0 PL=0
MOVL C01123 V=800.0 PL=0
MOVL C01124 V=800.0 PL=0
MOVL C01125 V=800.0 PL=0
MOVL C01126 V=800.0 PL=0
MOVL C01127 V=800.0 PL=0
MOVL C01128 V=800.0 PL=0
MOVL C01129 V=800.0 PL=0
MOVL C01130 V=800.0 PL=0
MOVL C01131 V=800.0 PL=0
MOVL C01132 V=800.0 PL=0
MOVL C01133 V=800.0 PL=0
MOVL C01134 V=800.0 PL=0
MOVL C01135 V=800.0 PL=0
MOVL C01136 V=800.0 PL=0
MOVL C01137 V=800.0 PL=0
MOVL C01138 V=800.0 PL=0
MOVL C01139 V=800.0 PL=0
MOVL C01140 V=800.0 PL=0
MOVL C01141 V=800.0 PL=0
MOVL C01142 V=800.0 PL=0
MOVL C01143 V=800.0 PL=0
MOVL C01144 V=800.0 PL=0
MOVL C01145 V=800.0 PL=0
MOVL C01146 V=800.0 PL=0
MOVL C01147 V=800.0 PL=0
MOVL C01148 V=800.0 PL=0
MOVL C01149 V=800.0 PL=0
MOVL C01150 V=800.0 PL=0
MOVL C01151 V=800.0 PL=0
MOVL C01152 V=800.0 PL=0
MOVL C01153 V=800.0 PL=0
MOVL C01154 V=800.0 PL=0
MOVL C01155 V=800.0 PL=0
MOVL C01156 V=800.0 PL=0
MOVL C01157 V=800.0 PL=0
MOVL C01158 V=800.0 PL=0
MOVL C01159 V=800.0 PL=0
MOVL C01160 V=800.0 PL=0
MOVL C01161 V=800.0 PL=0
MOVL C01162 V=800.0 PL=0
MOVL C01163 V=800.0 PL=0
MOVL C01164 V=800.0 PL=0
MOVL C01165 V=800.0 PL=0
MOVL C01166 V=800.0 PL=0
MOVL C01167 V=800.0 PL=0
MOVL C01168 V=800.0 PL=0
MOVL C01169 V=800.0 PL=0
MOVL C01170 V=800.0 PL=0
MOVL C01171 V=800.0 PL=0
MOVL C01172 V=800.0 PL=0
MOVL C01173 V=800.0 PL=0
MOVL C01174 V=800.0 PL=0
MOVL C01175 V=800.0 PL=0
MOVL C01176 V=800.0 PL=0
MOVL C01177 V=800.0 PL=0
MOVL C01178 V=800.0 PL=0
MOVL C01179 V=800.0 PL=0
MOVL C01180 V=800.0 PL=0
MOVL C01181 V=800.0 PL=0
MOVL C01182 V=800.0 PL=0
MOVL C01183 V=800.0 PL=0
MOVL C01184 V=800.0 PL=0
MOVL C01185 V=800.0 PL=0
MOVL C01186 V=800.0 PL=0
MOVL C01187 V=800.0 PL=0
MOVL C01188 V=800.0 PL=0
MOVL C01189 V=800.0 PL=0
MOVL C01190 V=800.0 PL=0
MOVL C01191 V=800.0 PL=0
MOVL C01192 V=800.0 PL=0
MOVL C01193 V=800.0 PL=0
MOVL C01194 V=800.0 PL=0
MOVL C01195 V=800.0 PL=0
MOVL C01196 V=800.0 PL=0
MOVL C01197 V=800.0 PL=0
MOVL C01198 V=800.0 PL=0
MOVL C01199 V=800.0 PL=0
MOVL C01200 V=800.0 PL=0
MOVL C01201 V=800.0 PL=0
MOVL C01202 V=800.0 PL=0
MOVL C01203 V=800.0 PL=0
MOVL C01204 V=800.0 PL=0
MOVL C01205 V=800.0 PL=0
MOVL C01206 V=800.0 PL=0
MOVL C01207 V=800.0 PL=0
MOVL C01208 V=800.0 PL=0
MOVL C01209 V=800.0 PL=0
MOVL C01210 V=800.0 PL=0
MOVL C01211 V=800.0 PL=0
MOVL C01212 V=800.0 PL=0
MOVL C01213 V=800.0 PL=0
MOVL C01214 V=800.0 PL=0
MOVL C01215 V=800.0 PL=0
MOVL C01216 V=800.0 PL=0
MOVL C01217 V=800.0 PL=0
MOVL C01218 V=800.0 PL=0
MOVL C01219 V=800.0 PL=0
MOVL C01220 V=800.0 PL=0
MOVL C01221 V=800.0 PL=0
MOVL C01222 V=800.0 PL=0
MOVL C01223 V=800.0 PL=0
MOVL C01224 V=800.0 PL=0
MOVL C01225 V=800.0 PL=0
MOVL C01226 V=800.0 PL=0
MOVL C01227 V=800.0 PL=0
MOVL C01228 V=800.0 PL=0
MOVL C01229 V=800.0 PL=0
MOVL C01230 V=800.0 PL=0
MOVL C01231 V=800.0 PL=0
MOVL C01232 V=800.0 PL=0
MOVL C01233 V=800.0 PL=0
MOVL C01234 V=800.0 PL=0
MOVL C01235 V=800.0 PL=0
MOVL C01236 V=800.0 PL=0
MOVL C01237 V=800.0 PL=0
MOVL C01238 V=800.0 PL=0
MOVL C01239 V=800.0 PL=0
MOVL C01240 V=800.0 PL=0
MOVL C01241 V=800.0 PL=0
MOVL C01242 V=800.0 PL=0
MOVL C01243 V=800.0 PL=0
MOVL C01244 V=800.0 PL=0
MOVL C01245 V=800.0 PL=0
MOVL C01246 V=800.0 PL=0
MOVL C01247 V=800.0 PL=0
MOVL C01248 V=800.0 PL=0
MOVL C01249 V=800.0 PL=0
MOVL C01250 V=800.0 PL=0
MOVL C01251 V=800.0 PL=0
MOVL C01252 V=800.0 PL=0
MOVL C01253 V=800.0 PL=0
MOVL C01254 V=800.0 PL=0
MOVL C01255 V=800.0 PL=0
MOVL C01256 V=800.0 PL=0
MOVL C01257 V=800.0 PL=0
MOVL C01258 V=800.0 PL=0
MOVL C01259 V=800.0 PL=0
MOVL C01260 V=800.0 PL=0
MOVL C01261 V=800.0 PL=0
MOVL C01262 V=800.0 PL=0
MOVL C01263 V=800.0 PL=0
MOVL C01264 V=800.0 PL=0
MOVL C01265 V=800.0 PL=0
MOVL C01266 V=800.0 PL=0
MOVL C01267 V=800.0 PL=0
MOVL C01268 V=800.0 PL=0
MOVL C01269 V=800.0 PL=0
MOVL C01270 V=800.0 PL=0
MOVL C01271 V=800.0 PL=0
MOVL C01272 V=800.0 PL=0
MOVL C01273 V=800.0 PL=0
MOVL C01274 V=800.0 PL=0
MOVL C01275 V=800.0 PL=0
MOVL C01276 V=800.0 PL=0
MOVL C01277 V=800.0 PL=0
MOVL C01278 V=800.0 PL=0
MOVL C01279 V=800.0 PL=0
MOVL C01280 V=800.0 PL=0
MOVL C01281 V=800.0 PL=0
MOVL C01282 V=800.0 PL=0
MOVL C01283 V=800.0 PL=0
MOVL C01284 V=800.0 PL=0
MOVL C01285 V=800.0 PL=0
MOVL C01286 V=800.0 PL=0
MOVL C01287 V=800.0 PL=0
MOVL C01288 V=800.0 PL=0
MOVL C01289 V=800.0 PL=0
MOVL C01290 V=800.0 PL=0
MOVL C01291 V=800.0 PL=0
MOVL C01292 V=800.0 PL=0
MOVL C01293 V=800.0 PL=0
MOVL C01294 V=800.0 PL=0
MOVL C01295 V=800.0 PL=0
MOVL C01296 V=800.0 PL=0
MOVL C01297 V=800.0 PL=0
MOVL C01298 V=800.0 PL=0
MOVL C01299 V=800.0 PL=0
MOVL C01300 V=800.0 PL=0
MOVL C01301 V=800.0 PL=0
MOVL C01302 V=800.0 PL=0
MOVL C01303 V=800.0 PL=0
MOVL C01304 V=800.0 PL=0
MOVL C01305 V=800.0 PL=0
MOVL C01306 V=800.0 PL=0
MOVL C01307 V=800.0 PL=0
MOVL C01308 V=800.0 PL=0
MOVL C01309 V=800.0 PL=0
MOVL C01310 V=800.0 PL=0
MOVL C01311 V=800.0 PL=0
MOVL C01312 V=800.0 PL=0
MOVL C01313 V=800.0 PL=0
MOVL C01314 V=800.0 PL=0
MOVL C01315 V=800.0 PL=0
MOVL C01316 V=800.0 PL=0
MOVL C01317 V=800.0 PL=0
MOVL C01318 V=800.0 PL=0
MOVL C01319 V=800.0 PL=0
MOVL C01320 V=800.0 PL=0
MOVL C01321 V=800.0 PL=0
MOVL C01322 V=800.0 PL=0
MOVL C01323 V=800.0 PL=0
MOVL C01324 V=800.0 PL=0
MOVL C01325 V=800.0 PL=0
MOVL C01326 V=800.0 PL=0
MOVL C01327 V=800.0 PL=0
MOVL C01328 V=800.0 PL=0
MOVL C01329 V=800.0 PL=0
MOVL C01330 V=800.0 PL=0
MOVL C01331 V=800.0 PL=0
MOVL C01332 V=800.0 PL=0
MOVL C01333 V=800.0 PL=0
MOVL C01334 V=800.0 PL=0
MOVL C01335 V=800.0 PL=0
MOVL C01336 V=800.0 PL=0
MOVL C01337 V=800.0 PL=0
MOVL C01338 V=800.0 PL=0
MOVL C01339 V=800.0 PL=0
MOVL C01340 V=800.0 PL=0
MOVL C01341 V=800.0 PL=0
MOVL C01342 V=800.0 PL=0
MOVL C01343 V=800.0 PL=0
MOVL C01344 V=800.0 PL=0
MOVL C01345 V=800.0 PL=0
MOVL C01346 V=800.0 PL=0
MOVL C01347 V=800.0 PL=0
MOVL C01348 V=800.0 PL=0
MOVL C01349 V=800.0 PL=0
MOVL C01350 V=800.0 PL=0
MOVL C01351 V=800.0 PL=0
MOVL C01352 V=800.0 PL=0
MOVL C01353 V=800.0 PL=0
MOVL C01354 V=800.0 PL=0
MOVL C01355 V=800.0 PL=0
MOVL C01356 V=800.0 PL=0
MOVL C01357 V=800.0 PL=0
MOVL C01358 V=800.0 PL=0
MOVL C01359 V=800.0 PL=0
MOVL C01360 V=800.0 PL=0
MOVL C01361 V=800.0 PL=0
MOVL C01362 V=800.0 PL=0
MOVL C01363 V=800.0 PL=0
MOVL C01364 V=800.0 PL=0
MOVL C01365 V=800.0 PL=0
MOVL C01366 V=800.0 PL=0
MOVL C01367 V=800.0 PL=0
MOVL C01368 V=800.0 PL=0
MOVL C01369 V=800.0 PL=0
MOVL C01370 V=800.0 PL=0
MOVL C01371 V=800.0 PL=0
MOVL C01372 V=800.0 PL=0
MOVL C01373 V=800.0 PL=0
MOVL C01374 V=800.0 PL=0
MOVL C01375 V=800.0 PL=0
MOVL C01376 V=800.0 PL=0
MOVL C01377 V=800.0 PL=0
MOVL C01378 V=800.0 PL=0
MOVL C01379 V=800.0 PL=0
MOVL C01380 V=800.0 PL=0
MOVL C01381 V=800.0 PL=0
MOVL C01382 V=800.0 PL=0
MOVL C01383 V=800.0 PL=0
MOVL C01384 V=800.0 PL=0
MOVL C01385 V=800.0 PL=0
MOVL C01386 V=800.0 PL=0
MOVL C01387 V=800.0 PL=0
MOVL C01388 V=800.0 PL=0
MOVL C01389 V=800.0 PL=0
MOVL C01390 V=800.0 PL=0
MOVL C01391 V=800.0 PL=0
MOVL C01392 V=800.0 PL=0
MOVL C01393 V=800.0 PL=0
MOVL C01394 V=800.0 PL=0
MOVL C01395 V=800.0 PL=0
MOVL C01396 V=800.0 PL=0
MOVL C01397 V=800.0 PL=0
MOVL C01398 V=800.0 PL=0
MOVL C01399 V=800.0 PL=0
MOVL C01400 V=800.0 PL=0
MOVL C01401 V=800.0 PL=0
MOVL C01402 V=800.0 PL=0
MOVL C01403 V=800.0 PL=0
MOVL C01404 V=800.0 PL=0
MOVL C01405 V=800.0 PL=0
MOVL C01406 V=800.0 PL=0
MOVL C01407 V=800.0 PL=0
MOVL C01408 V=800.0 PL=0
MOVL C01409 V=800.0 PL=0
MOVL C01410 V=800.0 PL=0
MOVL C01411 V=800.0 PL=0
MOVL C01412 V=800.0 PL=0
MOVL C01413 V=800.0 PL=0
MOVL C01414 V=800.0 PL=0
MOVL C01415 V=800.0 PL=0
MOVL C01416 V=800.0 PL=0
MOVL C01417 V=800.0 PL=0
MOVL C01418 V=800.0 PL=0
MOVL C01419 V=800.0 PL=0
MOVL C01420 V=800.0 PL=0
MOVL C01421 V=800.0 PL=0
MOVL C01422 V=800.0 PL=0
MOVL C01423 V=800.0 PL=0
MOVL C01424 V=800.0 PL=0
MOVL C01425 V=800.0 PL=0
MOVL C01426 V=800.0 PL=0
MOVL C01427 V=800.0 PL=0
MOVL C01428 V=800.0 PL=0
MOVL C01429 V=800.0 PL=0
MOVL C01430 V=800.0 PL=0
MOVL C01431 V=800.0 PL=0
MOVL C01432 V=800.0 PL=0
MOVL C01433 V=800.0 PL=0
MOVL C01434 V=800.0 PL=0
MOVL C01435 V=800.0 PL=0
MOVL C01436 V=800.0 PL=0
MOVL C01437 V=800.0 PL=0
MOVL C01438 V=800.0 PL=0
MOVL C01439 V=800.0 PL=0
MOVL C01440 V=800.0 PL=0
MOVL C01441 V=800.0 PL=0
MOVL C01442 V=800.0 PL=0
MOVL C01443 V=800.0 PL=0
MOVL C01444 V=800.0 PL=0
MOVL C01445 V=800.0 PL=0
MOVL C01446 V=800.0 PL=0
MOVL C01447 V=800.0 PL=0
MOVL C01448 V=800.0 PL=0
MOVL C01449 V=800.0 PL=0
MOVL C01450 V=800.0 PL=0
MOVL C01451 V=800.0 PL=0
MOVL C01452 V=800.0 PL=0
MOVL C01453 V=800.0 PL=0
MOVL C01454 V=800.0 PL=0
MOVL C01455 V=800.0 PL=0
MOVL C01456 V=800.0 PL=0
MOVL C01457 V=800.0 PL=0
MOVL C01458 V=800.0 PL=0
MOVL C01459 V=800.0 PL=0
MOVL C01460 V=800.0 PL=0
MOVL C01461 V=800.0 PL=0
MOVL C01462 V=800.0 PL=0
MOVL C01463 V=800.0 PL=0
MOVL C01464 V=800.0 PL=0
MOVL C01465 V=800.0 PL=0
MOVL C01466 V=800.0 PL=0
MOVL C01467 V=800.0 PL=0
MOVL C01468 V=800.0 PL=0
MOVL C01469 V=800.0 PL=0
MOVL C01470 V=800.0 PL=0
MOVL C01471 V=800.0 PL=0
MOVL C01472 V=800.0 PL=0
MOVL C01473 V=800.0 PL=0
MOVL C01474 V=800.0 PL=0
MOVL C01475 V=800.0 PL=0
MOVL C01476 V=800.0 PL=0
MOVL C01477 V=800.0 PL=0
MOVL C01478 V=800.0 PL=0
MOVL C01479 V=800.0 PL=0
MOVL C01480 V=800.0 PL=0
MOVL C01481 V=800.0 PL=0
MOVL C01482 V=800.0 PL=0
MOVL C01483 V=800.0 PL=0
MOVL C01484 V=800.0 PL=0
MOVL C01485 V=800.0 PL=0
MOVL C01486 V=800.0 PL=0
MOVL C01487 V=800.0 PL=0
MOVL C01488 V=800.0 PL=0
MOVL C01489 V=800.0 PL=0
MOVL C01490 V=800.0 PL=0
MOVL C01491 V=800.0 PL=0
MOVL C01492 V=800.0 PL=0
MOVL C01493 V=800.0 PL=0
MOVL C01494 V=800.0 PL=0
MOVL C01495 V=800.0 PL=0
MOVL C01496 V=800.0 PL=0
MOVL C01497 V=800.0 PL=0
MOVL C01498 V=800.0 PL=0
MOVL C01499 V=800.0 PL=0
MOVL C01500 V=800.0 PL=0
MOVL C01501 V=800.0 PL=0
MOVL C01502 V=800.0 PL=0
MOVL C01503 V=800.0 PL=0
MOVL C01504 V=800.0 PL=0
MOVL C01505 V=800.0 PL=0
MOVL C01506 V=800.0 PL=0
MOVL C01507 V=800.0 PL=0
MOVL C01508 V=800.0 PL=0
MOVL C01509 V=800.0 PL=0
MOVL C01510 V=800.0 PL=0
MOVL C01511 V=800.0 PL=0
MOVL C01512 V=800.0 PL=0
MOVL C01513 V=800.0 PL=0
MOVL C01514 V=800.0 PL=0
MOVL C01515 V=800.0 PL=0
MOVL C01516 V=800.0 PL=0
MOVL C01517 V=800.0 PL=0
MOVL C01518 V=800.0 PL=0
MOVL C01519 V=800.0 PL=0
MOVL C01520 V=800.0 PL=0
MOVL C01521 V=800.0 PL=0
MOVL C01522 V=800.0 PL=0
MOVL C01523 V=800.0 PL=0
MOVL C01524 V=800.0 PL=0
MOVL C01525 V=800.0 PL=0
MOVL C01526 V=800.0 PL=0
MOVL C01527 V=800.0 PL=0
MOVL C01528 V=800.0 PL=0
MOVL C01529 V=800.0 PL=0
MOVL C01530 V=800.0 PL=0
MOVL C01531 V=800.0 PL=0
MOVL C01532 V=800.0 PL=0
MOVL C01533 V=800.0 PL=0
MOVL C01534 V=800.0 PL=0
MOVL C01535 V=800.0 PL=0
MOVL C01536 V=800.0 PL=0
MOVL C01537 V=800.0 PL=0
MOVL C01538 V=800.0 PL=0
MOVL C01539 V=800.0 PL=0
MOVL C01540 V=800.0 PL=0
MOVL C01541 V=800.0 PL=0
MOVL C01542 V=800.0 PL=0
MOVL C01543 V=800.0 PL=0
MOVL C01544 V=800.0 PL=0
MOVL C01545 V=800.0 PL=0
MOVL C01546 V=800.0 PL=0
MOVL C01547 V=800.0 PL=0
MOVL C01548 V=800.0 PL=0
MOVL C01549 V=800.0 PL=0
MOVL C01550 V=800.0 PL=0
MOVL C01551 V=800.0 PL=0
MOVL C01552 V=800.0 PL=0
MOVL C01553 V=800.0 PL=0
MOVL C01554 V=800.0 PL=0
MOVL C01555 V=800.0 PL=0
MOVL C01556 V=800.0 PL=0
MOVL C01557 V=800.0 PL=0
MOVL C01558 V=800.0 PL=0
MOVL C01559 V=800.0 PL=0
MOVL C01560 V=800.0 PL=0
MOVL C01561 V=800.0 PL=0
MOVL C01562 V=800.0 PL=0
MOVL C01563 V=800.0 PL=0
MOVL C01564 V=800.0 PL=0
MOVL C01565 V=800.0 PL=0
MOVL C01566 V=800.0 PL=0
MOVL C01567 V=800.0 PL=0
MOVL C01568 V=800.0 PL=0
MOVL C01569 V=800.0 PL=0
MOVL C01570 V=800.0 PL=0
MOVL C01571 V=800.0 PL=0
MOVL C01572 V=800.0 PL=0
MOVL C01573 V=800.0 PL=0
MOVL C01574 V=800.0 PL=0
MOVL C01575 V=800.0 PL=0
MOVL C01576 V=800.0 PL=0
MOVL C01577 V=800.0 PL=0
MOVL C01578 V=800.0 PL=0
MOVL C01579 V=800.0 PL=0
MOVL C01580 V=800.0 PL=0
MOVL C01581 V=800.0 PL=0
MOVL C01582 V=800.0 PL=0
MOVL C01583 V=800.0 PL=0
MOVL C01584 V=800.0 PL=0
MOVL C01585 V=800.0 PL=0
MOVL C01586 V=800.0 PL=0
MOVL C01587 V=800.0 PL=0
MOVL C01588 V=800.0 PL=0
MOVL C01589 V=800.0 PL=0
MOVL C01590 V=800.0 PL=0
MOVL C01591 V=800.0 PL=0
MOVL C01592 V=800.0 PL=0
MOVL C01593 V=800.0 PL=0
MOVL C01594 V=800.0 PL=0
MOVL C01595 V=800.0 PL=0
MOVL C01596 V=800.0 PL=0
MOVL C01597 V=800.0 PL=0
MOVL C01598 V=800.0 PL=0
MOVL C01599 V=800.0 PL=0
MOVL C01600 V=800.0 PL=0
MOVL C01601 V=800.0 PL=0
MOVL C01602 V=800.0 PL=0
MOVL C01603 V=800.0 PL=0
MOVL C01604 V=800.0 PL=0
MOVL C01605 V=800.0 PL=0
MOVL C01606 V=800.0 PL=0
MOVL C01607 V=800.0 PL=0
MOVL C01608 V=800.0 PL=0
MOVL C01609 V=800.0 PL=0
MOVL C01610 V=800.0 PL=0
MOVL C01611 V=800.0 PL=0
MOVL C01612 V=800.0 PL=0
MOVL C01613 V=800.0 PL=0
MOVL C01614 V=800.0 PL=0
MOVL C01615 V=800.0 PL=0
MOVL C01616 V=800.0 PL=0
MOVL C01617 V=800.0 PL=0
MOVL C01618 V=800.0 PL=0
MOVL C01619 V=800.0 PL=0
MOVL C01620 V=800.0 PL=0
MOVL C01621 V=800.0 PL=0
MOVL C01622 V=800.0 PL=0
MOVL C01623 V=800.0 PL=0
MOVL C01624 V=800.0 PL=0
MOVL C01625 V=800.0 PL=0
MOVL C01626 V=800.0 PL=0
MOVL C01627 V=800.0 PL=0
MOVL C01628 V=800.0 PL=0
MOVL C01629 V=800.0 PL=0
MOVL C01630 V=800.0 PL=0
MOVL C01631 V=800.0 PL=0
MOVL C01632 V=800.0 PL=0
MOVL C01633 V=800.0 PL=0
MOVL C01634 V=800.0 PL=0
MOVL C01635 V=800.0 PL=0
MOVL C01636 V=800.0 PL=0
MOVL C01637 V=800.0 PL=0
MOVL C01638 V=800.0 PL=0
MOVL C01639 V=800.0 PL=0
MOVL C01640 V=800.0 PL=0
MOVL C01641 V=800.0 PL=0
MOVL C01642 V=800.0 PL=0
MOVL C01643 V=800.0 PL=0
MOVL C01644 V=800.0 PL=0
MOVL C01645 V=800.0 PL=0
MOVL C01646 V=800.0 PL=0
MOVL C01647 V=800.0 PL=0
MOVL C01648 V=800.0 PL=0
MOVL C01649 V=800.0 PL=0
MOVL C01650 V=800.0 PL=0
MOVL C01651 V=800.0 PL=0
MOVL C01652 V=800.0 PL=0
MOVL C01653 V=800.0 PL=0
MOVL C01654 V=800.0 PL=0
MOVL C01655 V=800.0 PL=0
MOVL C01656 V=800.0 PL=0
MOVL C01657 V=800.0 PL=0
MOVL C01658 V=800.0 PL=0
MOVL C01659 V=800.0 PL=0
MOVL C01660 V=800.0 PL=0
MOVL C01661 V=800.0 PL=0
MOVL C01662 V=800.0 PL=0
MOVL C01663 V=800.0 PL=0
MOVL C01664 V=800.0 PL=0
MOVL C01665 V=800.0 PL=0
MOVL C01666 V=800.0 PL=0
MOVL C01667 V=800.0 PL=0
MOVL C01668 V=800.0 PL=0
MOVL C01669 V=800.0 PL=0
MOVL C01670 V=800.0 PL=0
MOVL C01671 V=800.0 PL=0
MOVL C01672 V=800.0 PL=0
MOVL C01673 V=800.0 PL=0
MOVL C01674 V=800.0 PL=0
MOVL C01675 V=800.0 PL=0
MOVL C01676 V=800.0 PL=0
MOVL C01677 V=800.0 PL=0
MOVL C01678 V=800.0 PL=0
MOVL C01679 V=800.0 PL=0
MOVL C01680 V=800.0 PL=0
MOVL C01681 V=800.0 PL=0
MOVL C01682 V=800.0 PL=0
MOVL C01683 V=800.0 PL=0
MOVL C01684 V=800.0 PL=0
MOVL C01685 V=800.0 PL=0
MOVL C01686 V=800.0 PL=0
MOVL C01687 V=800.0 PL=0
MOVL C01688 V=800.0 PL=0
MOVL C01689 V=800.0 PL=0
MOVL C01690 V=800.0 PL=0
MOVL C01691 V=800.0 PL=0
MOVL C01692 V=800.0 PL=0
MOVL C01693 V=800.0 PL=0
MOVL C01694 V=800.0 PL=0
MOVL C01695 V=800.0 PL=0
MOVL C01696 V=800.0 PL=0
MOVL C01697 V=800.0 PL=0
MOVL C01698 V=800.0 PL=0
MOVL C01699 V=800.0 PL=0
MOVL C01700 V=800.0 PL=0
MOVL C01701 V=800.0 PL=0
MOVL C01702 V=800.0 PL=0
MOVL C01703 V=800.0 PL=0
MOVL C01704 V=800.0 PL=0
MOVL C01705 V=800.0 PL=0
MOVL C01706 V=800.0 PL=0
MOVL C01707 V=800.0 PL=0
MOVL C01708 V=800.0 PL=0
MOVL C01709 V=800.0 PL=0
MOVL C01710 V=800.0 PL=0
MOVL C01711 V=800.0 PL=0
MOVL C01712 V=800.0 PL=0
MOVL C01713 V=800.0 PL=0
MOVL C01714 V=800.0 PL=0
MOVL C01715 V=800.0 PL=0
MOVL C01716 V=800.0 PL=0
MOVL C01717 V=800.0 PL=0
MOVL C01718 V=800.0 PL=0
MOVL C01719 V=800.0 PL=0
MOVL C01720 V=800.0 PL=0
MOVL C01721 V=800.0 PL=0
MOVL C01722 V=800.0 PL=0
MOVL C01723 V=800.0 PL=0
MOVL C01724 V=800.0 PL=0
MOVL C01725 V=800.0 PL=0
MOVL C01726 V=800.0 PL=0
MOVL C01727 V=800.0 PL=0
MOVL C01728 V=800.0 PL=0
MOVL C01729 V=800.0 PL=0
MOVL C01730 V=800.0 PL=0
MOVL C01731 V=800.0 PL=0
MOVL C01732 V=800.0 PL=0
MOVL C01733 V=800.0 PL=0
MOVL C01734 V=800.0 PL=0
MOVL C01735 V=800.0 PL=0
MOVL C01736 V=800.0 PL=0
MOVL C01737 V=800.0 PL=0
MOVL C01738 V=800.0 PL=0
MOVL C01739 V=800.0 PL=0
MOVL C01740 V=800.0 PL=0
MOVL C01741 V=800.0 PL=0
MOVL C01742 V=800.0 PL=0
MOVL C01743 V=800.0 PL=0
MOVL C01744 V=800.0 PL=0
MOVL C01745 V=800.0 PL=0
MOVL C01746 V=800.0 PL=0
MOVL C01747 V=800.0 PL=0
MOVL C01748 V=800.0 PL=0
MOVL C01749 V=800.0 PL=0
MOVL C01750 V=800.0 PL=0
MOVL C01751 V=800.0 PL=0
MOVL C01752 V=800.0 PL=0
MOVL C01753 V=800.0 PL=0
MOVL C01754 V=800.0 PL=0
MOVL C01755 V=800.0 PL=0
MOVL C01756 V=800.0 PL=0
MOVL C01757 V=800.0 PL=0
MOVL C01758 V=800.0 PL=0
MOVL C01759 V=800.0 PL=0
MOVL C01760 V=800.0 PL=0
MOVL C01761 V=800.0 PL=0
MOVL C01762 V=800.0 PL=0
MOVL C01763 V=800.0 PL=0
MOVL C01764 V=800.0 PL=0
MOVL C01765 V=800.0 PL=0
MOVL C01766 V=800.0 PL=0
MOVL C01767 V=800.0 PL=0
MOVL C01768 V=800.0 PL=0
MOVL C01769 V=800.0 PL=0
MOVL C01770 V=800.0 PL=0
MOVL C01771 V=800.0 PL=0
MOVL C01772 V=800.0 PL=0
MOVL C01773 V=800.0 PL=0
MOVL C01774 V=800.0 PL=0
MOVL C01775 V=800.0 PL=0
MOVL C01776 V=800.0 PL=0
MOVL C01777 V=800.0 PL=0
MOVL C01778 V=800.0 PL=0
MOVL C01779 V=800.0 PL=0
MOVL C01780 V=800.0 PL=0
MOVL C01781 V=800.0 PL=0
MOVL C01782 V=800.0 PL=0
MOVL C01783 V=800.0 PL=0
MOVL C01784 V=800.0 PL=0
MOVL C01785 V=800.0 PL=0
MOVL C01786 V=800.0 PL=0
MOVL C01787 V=800.0 PL=0
MOVL C01788 V=800.0 PL=0
MOVL C01789 V=800.0 PL=0
MOVL C01790 V=800.0 PL=0
MOVL C01791 V=800.0 PL=0
MOVL C01792 V=800.0 PL=0
MOVL C01793 V=800.0 PL=0
MOVL C01794 V=800.0 PL=0
MOVL C01795 V=800.0 PL=0
MOVL C01796 V=800.0 PL=0
MOVL C01797 V=800.0 PL=0
MOVL C01798 V=800.0 PL=0
MOVL C01799 V=800.0 PL=0
MOVL C01800 V=800.0 PL=0
MOVL C01801 V=800.0 PL=0
MOVL C01802 V=800.0 PL=0
MOVL C01803 V=800.0 PL=0
MOVL C01804 V=800.0 PL=0
MOVL C01805 V=800.0 PL=0
MOVL C01806 V=800.0 PL=0
MOVL C01807 V=800.0 PL=0
MOVL C01808 V=800.0 PL=0
MOVL C01809 V=800.0 PL=0
MOVL C01810 V=800.0 PL=0
MOVL C01811 V=800.0 PL=0
MOVL C01812 V=800.0 PL=0
MOVL C01813 V=800.0 PL=0
MOVL C01814 V=800.0 PL=0
MOVL C01815 V=800.0 PL=0
MOVL C01816 V=800.0 PL=0
MOVL C01817 V=800.0 PL=0
MOVL C01818 V=800.0 PL=0
MOVL C01819 V=800.0 PL=0
MOVL C01820 V=800.0 PL=0
MOVL C01821 V=800.0 PL=0
MOVL C01822 V=800.0 PL=0
MOVL C01823 V=800.0 PL=0
MOVL C01824 V=800.0 PL=0
MOVL C01825 V=800.0 PL=0
MOVL C01826 V=800.0 PL=0
MOVL C01827 V=800.0 PL=0
MOVL C01828 V=800.0 PL=0
MOVL C01829 V=800.0 PL=0
MOVL C01830 V=800.0 PL=0
MOVL C01831 V=800.0 PL=0
MOVL C01832 V=800.0 PL=0
MOVL C01833 V=800.0 PL=0
MOVL C01834 V=800.0 PL=0
MOVL C01835 V=800.0 PL=0
MOVL C01836 V=800.0 PL=0
MOVL C01837 V=800.0 PL=0
MOVL C01838 V=800.0 PL=0
MOVL C01839 V=800.0 PL=0
MOVL C01840 V=800.0 PL=0
MOVL C01841 V=800.0 PL=0
MOVL C01842 V=800.0 PL=0
MOVL C01843 V=800.0 PL=0
MOVL C01844 V=800.0 PL=0
MOVL C01845 V=800.0 PL=0
MOVL C01846 V=800.0 PL=0
MOVL C01847 V=800.0 PL=0
MOVL C01848 V=800.0 PL=0
MOVL C01849 V=800.0 PL=0
MOVL C01850 V=800.0 PL=0
MOVL C01851 V=800.0 PL=0
MOVL C01852 V=800.0 PL=0
MOVL C01853 V=800.0 PL=0
MOVL C01854 V=800.0 PL=0
MOVL C01855 V=800.0 PL=0
MOVL C01856 V=800.0 PL=0
MOVL C01857 V=800.0 PL=0
MOVL C01858 V=800.0 PL=0
MOVL C01859 V=800.0 PL=0
MOVL C01860 V=800.0 PL=0
MOVL C01861 V=800.0 PL=0
MOVL C01862 V=800.0 PL=0
MOVL C01863 V=800.0 PL=0
MOVL C01864 V=800.0 PL=0
MOVL C01865 V=800.0 PL=0
MOVL C01866 V=800.0 PL=0
MOVL C01867 V=800.0 PL=0
MOVL C01868 V=800.0 PL=0
MOVL C01869 V=800.0 PL=0
MOVL C01870 V=800.0 PL=0
MOVL C01871 V=800.0 PL=0
MOVL C01872 V=800.0 PL=0
MOVL C01873 V=800.0 PL=0
MOVL C01874 V=800.0 PL=0
MOVL C01875 V=800.0 PL=0
MOVL C01876 V=800.0 PL=0
MOVL C01877 V=800.0 PL=0
MOVL C01878 V=800.0 PL=0
MOVL C01879 V=800.0 PL=0
MOVL C01880 V=800.0 PL=0
MOVL C01881 V=800.0 PL=0
MOVL C01882 V=800.0 PL=0
MOVL C01883 V=800.0 PL=0
MOVL C01884 V=800.0 PL=0
MOVL C01885 V=800.0 PL=0
MOVL C01886 V=800.0 PL=0
MOVL C01887 V=800.0 PL=0
MOVL C01888 V=800.0 PL=0
MOVL C01889 V=800.0 PL=0
MOVL C01890 V=800.0 PL=0
MOVL C01891 V=800.0 PL=0
MOVL C01892 V=800.0 PL=0
MOVL C01893 V=800.0 PL=0
MOVL C01894 V=800.0 PL=0
MOVL C01895 V=800.0 PL=0
MOVL C01896 V=800.0 PL=0
MOVL C01897 V=800.0 PL=0
MOVL C01898 V=800.0 PL=0
MOVL C01899 V=800.0 PL=0
MOVL C01900 V=800.0 PL=0
MOVL C01901 V=800.0 PL=0
MOVL C01902 V=800.0 PL=0
MOVL C01903 V=800.0 PL=0
MOVL C01904 V=800.0 PL=0
MOVL C01905 V=800.0 PL=0
MOVL C01906 V=800.0 PL=0
MOVL C01907 V=800.0 PL=0
MOVL C01908 V=800.0 PL=0
MOVL C01909 V=800.0 PL=0
MOVL C01910 V=800.0 PL=0
MOVL C01911 V=800.0 PL=0
MOVL C01912 V=800.0 PL=0
MOVL C01913 V=800.0 PL=0
MOVL C01914 V=800.0 PL=0
MOVL C01915 V=800.0 PL=0
MOVL C01916 V=800.0 PL=0
MOVL C01917 V=800.0 PL=0
MOVL C01918 V=800.0 PL=0
MOVL C01919 V=800.0 PL=0
MOVL C01920 V=800.0 PL=0
MOVL C01921 V=800.0 PL=0
MOVL C01922 V=800.0 PL=0
MOVL C01923 V=800.0 PL=0
MOVL C01924 V=800.0 PL=0
MOVL C01925 V=800.0 PL=0
MOVL C01926 V=800.0 PL=0
MOVL C01927 V=800.0 PL=0
MOVL C01928 V=800.0 PL=0
MOVL C01929 V=800.0 PL=0
MOVL C01930 V=800.0 PL=0
MOVL C01931 V=800.0 PL=0
MOVL C01932 V=800.0 PL=0
MOVL C01933 V=800.0 PL=0
MOVL C01934 V=800.0 PL=0
MOVL C01935 V=800.0 PL=0
MOVL C01936 V=800.0 PL=0
MOVL C01937 V=800.0 PL=0
MOVL C01938 V=800.0 PL=0
MOVL C01939 V=800.0 PL=0
MOVL C01940 V=800.0 PL=0
MOVL C01941 V=800.0 PL=0
MOVL C01942 V=800.0 PL=0
MOVL C01943 V=800.0 PL=0
MOVL C01944 V=800.0 PL=0
MOVL C01945 V=800.0 PL=0
MOVL C01946 V=800.0 PL=0
MOVL C01947 V=800.0 PL=0
MOVL C01948 V=800.0 PL=0
MOVL C01949 V=800.0 PL=0
MOVL C01950 V=800.0 PL=0
MOVL C01951 V=800.0 PL=0
MOVL C01952 V=800.0 PL=0
MOVL C01953 V=800.0 PL=0
MOVL C01954 V=800.0 PL=0
MOVL C01955 V=800.0 PL=0
MOVL C01956 V=800.0 PL=0
MOVL C01957 V=800.0 PL=0
MOVL C01958 V=800.0 PL=0
MOVL C01959 V=800.0 PL=0
MOVL C01960 V=800.0 PL=0
MOVL C01961 V=800.0 PL=0
MOVL C01962 V=800.0 PL=0
MOVL C01963 V=800.0 PL=0
MOVL C01964 V=800.0 PL=0
MOVL C01965 V=800.0 PL=0
MOVL C01966 V=800.0 PL=0
MOVL C01967 V=800.0 PL=0
MOVL C01968 V=800.0 PL=0
MOVL C01969 V=800.0 PL=0
MOVL C01970 V=800.0 PL=0
MOVL C01971 V=800.0 PL=0
MOVL C01972 V=800.0 PL=0
MOVL C01973 V=800.0 PL=0
MOVL C01974 V=800.0 PL=0
MOVL C01975 V=800.0 PL=0
MOVL C01976 V=800.0 PL=0
MOVL C01977 V=800.0 PL=0
MOVL C01978 V=800.0 PL=0
MOVL C01979 V=800.0 PL=0
MOVL C01980 V=800.0 PL=0
MOVL C01981 V=800.0 PL=0
MOVL C01982 V=800.0 PL=0
MOVL C01983 V=800.0 PL=0
MOVL C01984 V=800.0 PL=0
MOVL C01985 V=800.0 PL=0
MOVL C01986 V=800.0 PL=0
MOVL C01987 V=800.0 PL=0
MOVL C01988 V=800.0 PL=0
MOVL C01989 V=800.0 PL=0
MOVL C01990 V=800.0 PL=0
MOVL C01991 V=800.0 PL=0
MOVL C01992 V=800.0 PL=0
MOVL C01993 V=800.0 PL=0
MOVL C01994 V=800.0 PL=0
MOVL C01995 V=800.0 PL=0
MOVL C01996 V=800.0 PL=0
MOVL C01997 V=800.0 PL=0
MOVL C01998 V=800.0 PL=0
MOVL C01999 V=800.0 PL=0
MOVL C02000 V=800.0 PL=0
MOVL C02001 V=800.0 PL=0
MOVL C02002 V=800.0 PL=0
MOVL C02003 V=800.0 PL=0
MOVL C02004 V=800.0 PL=0
MOVL C02005 V=800.0 PL=0
MOVL C02006 V=800.0 PL=0
MOVL C02007 V=800.0 PL=0
MOVL C02008 V=800.0 PL=0
MOVL C02009 V=800.0 PL=0
MOVL C02010 V=800.0 PL=0
MOVL C02011 V=800.0 PL=0
MOVL C02012 V=800.0 PL=0
MOVL C02013 V=800.0 PL=0
MOVL C02014 V=800.0 PL=0
MOVL C02015 V=800.0 PL=0
MOVL C02016 V=800.0 PL=0
MOVL C02017 V=800.0 PL=0
MOVL C02018 V=800.0 PL=0
MOVL C02019 V=800.0 PL=0
MOVL C02020 V=800.0 PL=0
MOVL C02021 V=800.0 PL=0
MOVL C02022 V=800.0 PL=0
MOVL C02023 V=800.0 PL=0
MOVL C02024 V=800.0 PL=0
MOVL C02025 V=800.0 PL=0
MOVL C02026 V=800.0 PL=0
MOVL C02027 V=800.0 PL=0
MOVL C02028 V=800.0 PL=0
MOVL C02029 V=800.0 PL=0
MOVL C02030 V=800.0 PL=0
MOVL C02031 V=800.0 PL=0
MOVL C02032 V=800.0 PL=0
MOVL C02033 V=800.0 PL=0
MOVL C02034 V=800.0 PL=0
MOVL C02035 V=800.0 PL=0
MOVL C02036 V=800.0 PL=0
MOVL C02037 V=800.0 PL=0
MOVL C02038 V=800.0 PL=0
MOVL C02039 V=800.0 PL=0
MOVL C02040 V=800.0 PL=0
MOVL C02041 V=800.0 PL=0
MOVL C02042 V=800.0 PL=0
MOVL C02043 V=800.0 PL=0
MOVL C02044 V=800.0 PL=0
MOVL C02045 V=800.0 PL=0
MOVL C02046 V=800.0 PL=0
MOVL C02047 V=800.0 PL=0
